C03653=1212.909,290.685,-66.684,-176.596,6.990,148.306
C03654=1212.913,290.437,-66.657,-176.598,6.987,148.306
C03655=1212.918,290.189,-66.627,-176.601,6.985,148.306
C03656=1212.922,289.941,-66.598,-176.603,6.983,148.306
C03657=1212.926,289.692,-66.569,-176.606,6.980,148.306
C03658=1212.931,289.418,-66.537,-176.609,6.977,148.306
C03659=1212.935,289.144,-66.505,-176.611,6.975,148.306
C03660=1212.940,288.869,-66.473,-176.614,6.972,148.306
C03661=1212.945,288.595,-66.442,-176.617,6.969,148.306
C03662=1212.950,288.347,-66.413,-176.619,6.967,148.306
C03663=1212.954,288.099,-66.384,-176.621,6.964,148.306
C03664=1212.958,287.851,-66.355,-176.624,6.962,148.307
C03665=1212.963,287.602,-66.327,-176.627,6.959,148.307
C03666=1212.967,287.354,-66.297,-176.629,6.957,148.307
C03667=1212.972,287.105,-66.268,-176.631,6.954,148.307
C03668=1212.976,286.858,-66.240,-176.634,6.952,148.307
C03669=1212.980,286.609,-66.211,-176.636,6.949,148.307
C03670=1212.985,286.360,-66.182,-176.639,6.946,148.307
C03671=1212.989,286.113,-66.154,-176.641,6.944,148.307
C03672=1212.993,285.864,-66.125,-176.644,6.941,148.307
C03673=1212.998,285.615,-66.096,-176.646,6.939,148.308
C03674=1213.002,285.368,-66.068,-176.648,6.937,148.308
C03675=1213.006,285.119,-66.039,-176.651,6.934,148.308
C03676=1213.011,284.870,-66.010,-176.654,6.932,148.308
C03677=1213.015,284.623,-65.982,-176.656,6.929,148.308
C03678=1213.019,284.374,-65.953,-176.658,6.927,148.308
C03679=1213.024,284.126,-65.925,-176.661,6.925,148.308
C03680=1213.028,283.878,-65.896,-176.664,6.922,148.308
C03681=1213.032,283.629,-65.867,-176.666,6.920,148.308
C03682=1213.037,283.381,-65.839,-176.668,6.918,148.308
C03683=1213.041,283.132,-65.811,-176.671,6.915,148.309
C03684=1213.045,282.884,-65.781,-176.673,6.913,148.309
C03685=1213.050,282.636,-65.754,-176.676,6.910,148.309
C03686=1213.054,282.387,-65.725,-176.679,6.908,148.309
C03687=1213.058,282.139,-65.697,-176.681,6.906,148.309
C03688=1213.063,281.890,-65.668,-176.683,6.903,148.309
C03689=1213.068,281.643,-65.639,-176.686,6.901,148.309
C03690=1213.071,281.394,-65.611,-176.689,6.898,148.309
C03691=1213.076,281.145,-65.582,-176.691,6.895,148.310
C03692=1213.080,280.898,-65.555,-176.693,6.894,148.310
C03693=1213.085,280.649,-65.526,-176.696,6.891,148.310
C03694=1213.089,280.401,-65.498,-176.698,6.888,148.310
C03695=1213.094,280.152,-65.469,-176.701,6.887,148.310
C03696=1213.098,279.905,-65.441,-176.704,6.883,148.310
C03697=1213.102,279.656,-65.412,-176.706,6.881,148.310
C03698=1213.106,279.408,-65.384,-176.709,6.879,148.311
C03699=1213.110,279.159,-65.356,-176.711,6.876,148.311
C03700=1213.115,278.911,-65.328,-176.713,6.874,148.311
C03701=1213.119,278.663,-65.300,-176.716,6.871,148.311
C03702=1213.124,278.414,-65.271,-176.718,6.869,148.311
C03703=1213.128,278.166,-65.243,-176.720,6.867,148.311
C03704=1213.132,277.917,-65.214,-176.724,6.864,148.311
C03705=1213.137,277.669,-65.187,-176.726,6.862,148.311
C03706=1213.141,277.420,-65.158,-176.728,6.860,148.311
C03707=1213.146,277.172,-65.130,-176.731,6.857,148.312
C03708=1213.149,276.924,-65.102,-176.733,6.855,148.312
C03709=1213.154,276.675,-65.074,-176.735,6.853,148.312
C03710=1213.159,276.428,-65.046,-176.738,6.850,148.312
C03711=1213.163,276.178,-65.018,-176.741,6.848,148.312
C03712=1213.168,275.930,-64.990,-176.744,6.845,148.312
C03713=1213.172,275.682,-64.962,-176.746,6.843,148.313
C03714=1213.177,275.433,-64.933,-176.748,6.841,148.313
C03715=1213.180,275.185,-64.905,-176.751,6.838,148.313
C03716=1213.185,274.937,-64.878,-176.753,6.836,148.313
C03717=1213.189,274.688,-64.849,-176.756,6.834,148.313
C03718=1213.194,274.440,-64.821,-176.759,6.831,148.313
C03719=1213.198,274.191,-64.794,-176.761,6.829,148.313
C03720=1213.202,273.943,-64.766,-176.763,6.827,148.314
C03721=1213.207,273.695,-64.737,-176.766,6.824,148.314
C03722=1213.211,273.446,-64.709,-176.769,6.822,148.314
C03723=1213.215,273.199,-64.682,-176.771,6.820,148.314
C03724=1213.220,272.949,-64.654,-176.773,6.817,148.314
C03725=1213.224,272.701,-64.626,-176.776,6.815,148.314
C03726=1213.228,272.453,-64.598,-176.778,6.813,148.314
C03727=1213.233,272.205,-64.570,-176.781,6.810,148.315
C03728=1213.238,271.956,-64.542,-176.784,6.808,148.315
C03729=1213.242,271.707,-64.514,-176.786,6.806,148.315
C03730=1213.246,271.459,-64.486,-176.788,6.804,148.315
C03731=1213.251,271.211,-64.459,-176.791,6.801,148.315
C03732=1213.255,270.962,-64.430,-176.794,6.799,148.315
C03733=1213.260,270.714,-64.403,-176.796,6.797,148.316
C03734=1213.264,270.465,-64.375,-176.799,6.794,148.316
C03735=1213.268,270.217,-64.347,-176.801,6.792,148.316
C03736=1213.272,269.969,-64.320,-176.804,6.790,148.316
C03737=1213.277,269.720,-64.292,-176.806,6.787,148.316
C03738=1213.281,269.472,-64.264,-176.808,6.785,148.316
C03739=1213.286,269.223,-64.237,-176.811,6.783,148.317
C03740=1213.290,268.975,-64.209,-176.814,6.780,148.317
C03741=1213.294,268.726,-64.182,-176.816,6.778,148.317
C03742=1213.299,268.478,-64.154,-176.818,6.776,148.317
C03743=1213.303,268.230,-64.126,-176.821,6.774,148.317
C03744=1213.308,267.981,-64.098,-176.824,6.771,148.317
C03745=1213.312,267.733,-64.070,-176.826,6.769,148.318
C03746=1213.316,267.484,-64.043,-176.829,6.767,148.318
C03747=1213.321,267.236,-64.015,-176.832,6.764,148.318
C03748=1213.325,266.988,-63.988,-176.834,6.762,148.318
C03749=1213.330,266.740,-63.960,-176.836,6.760,148.318
C03750=1213.334,266.491,-63.933,-176.839,6.758,148.318
C03751=1213.338,266.242,-63.906,-176.841,6.755,148.318
C03752=1213.343,265.994,-63.878,-176.844,6.753,148.319
C03753=1213.347,265.745,-63.851,-176.846,6.751,148.319
C03754=1213.351,265.497,-63.823,-176.849,6.748,148.319
C03755=1213.357,265.248,-63.795,-176.851,6.746,148.319
C03756=1213.361,265.000,-63.768,-176.854,6.744,148.319
C03757=1213.365,264.751,-63.740,-176.856,6.742,148.320
C03758=1213.370,264.503,-63.713,-176.859,6.739,148.320
C03759=1213.374,264.255,-63.685,-176.861,6.737,148.320
C03760=1213.379,264.006,-63.658,-176.864,6.735,148.320
C03761=1213.383,263.757,-63.631,-176.866,6.733,148.320
C03762=1213.387,263.485,-63.601,-176.869,6.730,148.321
C03763=1213.393,263.212,-63.571,-176.872,6.727,148.321
C03764=1213.397,262.940,-63.541,-176.875,6.725,148.321
C03765=1213.402,262.667,-63.511,-176.878,6.723,148.321
C03766=1213.406,262.418,-63.483,-176.880,6.721,148.321
C03767=1213.411,262.170,-63.456,-176.882,6.718,148.322
C03768=1213.416,261.921,-63.429,-176.886,6.716,148.322
C03769=1213.419,261.674,-63.402,-176.888,6.714,148.322
C03770=1213.424,261.425,-63.375,-176.890,6.712,148.322
C03771=1213.428,261.176,-63.347,-176.893,6.710,148.322
C03772=1213.433,260.927,-63.320,-176.896,6.707,148.323
C03773=1213.437,260.679,-63.292,-176.898,6.705,148.323
C03774=1213.442,260.431,-63.265,-176.900,6.703,148.323
C03775=1213.446,260.182,-63.238,-176.903,6.701,148.323
C03776=1213.450,259.933,-63.211,-176.906,6.698,148.323
C03777=1213.455,259.685,-63.184,-176.908,6.696,148.323
C03778=1213.459,259.437,-63.157,-176.910,6.694,148.324
C03779=1213.464,259.188,-63.130,-176.913,6.692,148.324
C03780=1213.468,258.940,-63.103,-176.915,6.690,148.324
C03781=1213.473,258.692,-63.075,-176.918,6.687,148.324
C03782=1213.477,258.443,-63.048,-176.921,6.685,148.324
C03783=1213.481,258.194,-63.021,-176.923,6.683,148.325
C03784=1213.485,257.946,-62.995,-176.925,6.681,148.325
C03785=1213.490,257.697,-62.967,-176.928,6.678,148.325
C03786=1213.495,257.449,-62.940,-176.931,6.676,148.325
C03787=1213.499,257.200,-62.913,-176.933,6.674,148.325
C03788=1213.504,256.952,-62.886,-176.936,6.672,148.326
C03789=1213.508,256.704,-62.860,-176.938,6.670,148.326
C03790=1213.512,256.455,-62.833,-176.941,6.667,148.326
C03791=1213.516,256.206,-62.805,-176.943,6.665,148.326
C03792=1213.521,255.957,-62.778,-176.946,6.663,148.326
C03793=1213.526,255.709,-62.751,-176.948,6.661,148.327
C03794=1213.530,255.461,-62.725,-176.951,6.658,148.327
C03795=1213.534,255.212,-62.698,-176.954,6.656,148.327
C03796=1213.539,254.964,-62.671,-176.956,6.654,148.327
C03797=1213.543,254.715,-62.645,-176.959,6.652,148.328
C03798=1213.548,254.467,-62.618,-176.961,6.650,148.328
C03799=1213.553,254.218,-62.591,-176.964,6.648,148.328
C03800=1213.557,253.970,-62.564,-176.967,6.646,148.328
C03801=1213.561,253.721,-62.537,-176.969,6.643,148.328
C03802=1213.566,253.473,-62.510,-176.971,6.642,148.329
C03803=1213.570,253.224,-62.483,-176.973,6.639,148.329
C03804=1213.574,252.976,-62.457,-176.977,6.637,148.329
C03805=1213.579,252.727,-62.430,-176.979,6.635,148.329
C03806=1213.584,252.479,-62.403,-176.981,6.633,148.329
C03807=1213.587,252.230,-62.376,-176.984,6.631,148.330
C03808=1213.592,251.981,-62.349,-176.986,6.629,148.330
C03809=1213.596,251.733,-62.323,-176.989,6.626,148.330
C03810=1213.601,251.484,-62.296,-176.992,6.624,148.330
C03811=1213.606,251.235,-62.269,-176.994,6.622,148.330
C03812=1213.609,250.987,-62.243,-176.997,6.620,148.331
C03813=1213.614,250.738,-62.217,-176.999,6.618,148.331
C03814=1213.618,250.490,-62.190,-177.001,6.616,148.331
C03815=1213.623,250.241,-62.163,-177.005,6.613,148.331
C03816=1213.628,249.993,-62.136,-177.007,6.611,148.331
C03817=1213.632,249.744,-62.110,-177.009,6.609,148.332
C03818=1213.637,249.496,-62.083,-177.012,6.607,148.332
C03819=1213.641,249.248,-62.057,-177.014,6.605,148.332
C03820=1213.646,248.999,-62.031,-177.017,6.603,148.332
C03821=1213.650,248.751,-62.004,-177.020,6.601,148.333
C03822=1213.655,248.502,-61.978,-177.022,6.598,148.333
C03823=1213.659,248.254,-61.951,-177.025,6.597,148.333
C03824=1213.663,248.005,-61.924,-177.027,6.595,148.333
C03825=1213.668,247.756,-61.899,-177.029,6.593,148.334
C03826=1213.672,247.508,-61.872,-177.032,6.591,148.334
C03827=1213.677,247.259,-61.846,-177.035,6.588,148.334
C03828=1213.681,247.010,-61.819,-177.037,6.586,148.334
C03829=1213.685,246.762,-61.792,-177.040,6.584,148.335
C03830=1213.690,246.513,-61.766,-177.042,6.582,148.335
C03831=1213.694,246.265,-61.740,-177.045,6.580,148.335
C03832=1213.699,246.016,-61.713,-177.047,6.578,148.335
C03833=1213.703,245.768,-61.687,-177.050,6.576,148.335
C03834=1213.708,245.519,-61.660,-177.053,6.573,148.336
C03835=1213.712,245.271,-61.634,-177.055,6.571,148.336
C03836=1213.717,245.022,-61.608,-177.057,6.569,148.336
C03837=1213.722,244.773,-61.582,-177.060,6.567,148.336
C03838=1213.725,244.525,-61.556,-177.063,6.565,148.337
C03839=1213.730,244.276,-61.529,-177.065,6.563,148.337
C03840=1213.734,244.028,-61.503,-177.067,6.561,148.337
C03841=1213.739,243.779,-61.477,-177.071,6.559,148.337
C03842=1213.743,243.530,-61.450,-177.073,6.557,148.338
C03843=1213.748,243.282,-61.425,-177.075,6.555,148.338
C03844=1213.753,243.033,-61.398,-177.078,6.553,148.338
C03845=1213.757,242.785,-61.372,-177.081,6.551,148.338
C03846=1213.761,242.536,-61.346,-177.083,6.549,148.338
C03847=1213.766,242.287,-61.320,-177.085,6.547,148.339
C03848=1213.770,242.039,-61.293,-177.088,6.545,148.339
C03849=1213.774,241.790,-61.268,-177.091,6.542,148.339
C03850=1213.780,241.542,-61.242,-177.093,6.540,148.339
C03851=1213.784,241.293,-61.215,-177.096,6.538,148.340
C03852=1213.788,241.045,-61.189,-177.098,6.536,148.340
C03853=1213.793,240.795,-61.163,-177.101,6.534,148.340
C03854=1213.797,240.547,-61.137,-177.103,6.532,148.341
C03855=1213.802,240.299,-61.111,-177.106,6.530,148.341
C03856=1213.806,240.050,-61.085,-177.108,6.528,148.341
C03857=1213.811,239.801,-61.059,-177.111,6.526,148.341
C03858=1213.815,239.552,-61.033,-177.114,6.524,148.342
C03859=1213.819,239.304,-61.007,-177.116,6.522,148.342
C03860=1213.824,239.056,-60.981,-177.119,6.520,148.342
C03861=1213.829,238.807,-60.955,-177.121,6.518,148.342
C03862=1213.833,238.558,-60.929,-177.124,6.516,148.343
C03863=1213.837,238.309,-60.904,-177.126,6.514,148.343
C03864=1213.842,238.061,-60.878,-177.129,6.512,148.343
C03865=1213.847,237.813,-60.851,-177.131,6.510,148.343
C03866=1213.851,237.541,-60.823,-177.135,6.507,148.344
C03867=1213.857,237.270,-60.795,-177.137,6.506,148.344
C03868=1213.861,236.999,-60.767,-177.140,6.503,148.344
C03869=1213.866,236.727,-60.739,-177.143,6.501,148.344
C03870=1213.871,236.478,-60.713,-177.145,6.499,148.345
C03871=1213.875,236.230,-60.688,-177.148,6.497,148.345
C03872=1213.879,235.981,-60.662,-177.150,6.495,148.345
C03873=1213.884,235.732,-60.635,-177.153,6.493,148.345
C03874=1213.889,235.484,-60.610,-177.155,6.491,148.346
C03875=1213.893,235.235,-60.584,-177.158,6.489,148.346
C03876=1213.897,234.986,-60.559,-177.160,6.487,148.346
C03877=1213.902,234.738,-60.533,-177.163,6.484,148.346
C03878=1213.906,234.489,-60.507,-177.166,6.482,148.347
C03879=1213.911,234.240,-60.482,-177.168,6.481,148.347
C03880=1213.915,233.992,-60.456,-177.171,6.479,148.347
C03881=1213.920,233.743,-60.431,-177.173,6.477,148.347
C03882=1213.925,233.494,-60.404,-177.176,6.475,148.348
C03883=1213.929,233.246,-60.378,-177.178,6.473,148.348
C03884=1213.934,232.997,-60.353,-177.181,6.471,148.348
C03885=1213.938,232.749,-60.327,-177.184,6.469,148.349
C03886=1213.942,232.500,-60.302,-177.186,6.467,148.349
C03887=1213.947,232.252,-60.276,-177.188,6.465,148.349
C03888=1213.951,232.003,-60.250,-177.191,6.463,148.349
C03889=1213.956,231.753,-60.225,-177.194,6.461,148.350
C03890=1213.961,231.505,-60.200,-177.196,6.459,148.350
C03891=1213.965,231.257,-60.174,-177.199,6.457,148.350
C03892=1213.970,231.008,-60.149,-177.202,6.455,148.350
C03893=1213.974,230.760,-60.123,-177.204,6.453,148.351
C03894=1213.978,230.511,-60.097,-177.207,6.451,148.351
C03895=1213.983,230.262,-60.073,-177.209,6.449,148.351
C03896=1213.987,230.013,-60.047,-177.212,6.447,148.352
C03897=1213.992,229.765,-60.021,-177.214,6.445,148.352
C03898=1213.996,229.516,-59.996,-177.217,6.443,148.352
C03899=1214.001,229.267,-59.971,-177.220,6.441,148.352
C03900=1214.006,229.019,-59.945,-177.222,6.439,148.353
C03901=1214.010,228.770,-59.920,-177.224,6.437,148.353
C03902=1214.014,228.521,-59.894,-177.227,6.436,148.353
C03903=1214.019,228.273,-59.869,-177.230,6.434,148.354
C03904=1214.023,228.024,-59.844,-177.232,6.432,148.354
C03905=1214.028,227.776,-59.819,-177.235,6.430,148.354
C03906=1214.032,227.527,-59.794,-177.237,6.428,148.354
C03907=1214.037,227.278,-59.768,-177.240,6.426,148.355
C03908=1214.041,227.030,-59.743,-177.242,6.424,148.355
C03909=1214.046,226.780,-59.717,-177.245,6.422,148.355
C03910=1214.051,226.532,-59.692,-177.248,6.420,148.356
C03911=1214.055,226.283,-59.666,-177.250,6.418,148.356
C03912=1214.059,226.035,-59.642,-177.253,6.416,148.356
C03913=1214.063,225.786,-59.617,-177.256,6.414,148.356
C03914=1214.069,225.537,-59.592,-177.258,6.412,148.357
C03915=1214.073,225.289,-59.566,-177.261,6.410,148.357
C03916=1214.078,225.040,-59.541,-177.263,6.408,148.357
C03917=1214.082,224.791,-59.516,-177.266,6.406,148.357
C03918=1214.086,224.543,-59.491,-177.268,6.404,148.358
C03919=1214.091,224.294,-59.466,-177.271,6.402,148.358
C03920=1214.096,224.046,-59.440,-177.273,6.400,148.358
C03921=1214.100,223.796,-59.415,-177.276,6.399,148.359
C03922=1214.105,223.548,-59.390,-177.279,6.397,148.359
C03923=1214.109,223.299,-59.366,-177.281,6.395,148.359
C03924=1214.114,223.051,-59.340,-177.284,6.393,148.359
C03925=1214.118,222.802,-59.315,-177.286,6.391,148.360
C03926=1214.123,222.553,-59.290,-177.289,6.389,148.360
C03927=1214.127,222.304,-59.265,-177.291,6.387,148.360
C03928=1214.132,222.056,-59.241,-177.294,6.385,148.361
C03929=1214.136,221.807,-59.215,-177.297,6.383,148.361
C03930=1214.141,221.558,-59.190,-177.299,6.382,148.361
C03931=1214.145,221.310,-59.165,-177.301,6.379,148.362
C03932=1214.150,221.061,-59.140,-177.304,6.378,148.362
C03933=1214.154,220.811,-59.115,-177.307,6.376,148.362
C03934=1214.158,220.564,-59.091,-177.309,6.374,148.363
C03935=1214.163,220.314,-59.066,-177.312,6.372,148.363
C03936=1214.168,220.066,-59.040,-177.315,6.370,148.363
C03937=1214.172,219.818,-59.016,-177.317,6.368,148.364
C03938=1214.177,219.568,-58.991,-177.320,6.366,148.364
C03939=1214.182,219.320,-58.966,-177.322,6.364,148.364
C03940=1214.185,219.071,-58.941,-177.325,6.362,148.364
C03941=1214.191,218.822,-58.917,-177.327,6.361,148.365
C03942=1214.195,218.573,-58.892,-177.330,6.359,148.365
C03943=1214.199,218.325,-58.867,-177.333,6.357,148.365
C03944=1214.204,218.076,-58.842,-177.335,6.355,148.366
C03945=1214.209,217.827,-58.817,-177.338,6.353,148.366
C03946=1214.213,217.579,-58.793,-177.341,6.351,148.366
C03947=1214.217,217.330,-58.767,-177.343,6.350,148.367
C03948=1214.222,217.081,-58.743,-177.346,6.348,148.367
C03949=1214.227,216.833,-58.718,-177.348,6.346,148.367
C03950=1214.231,216.583,-58.693,-177.351,6.344,148.367
C03951=1214.236,216.335,-58.669,-177.353,6.342,148.368
C03952=1214.241,216.087,-58.644,-177.356,6.340,148.368
C03953=1214.244,215.838,-58.620,-177.358,6.338,148.368
C03954=1214.250,215.589,-58.595,-177.361,6.336,148.369
C03955=1214.254,215.340,-58.571,-177.364,6.334,148.369
C03956=1214.259,215.091,-58.546,-177.366,6.333,148.369
C03957=1214.263,214.843,-58.522,-177.369,6.331,148.370
C03958=1214.267,214.593,-58.497,-177.372,6.329,148.370
C03959=1214.272,214.345,-58.473,-177.374,6.327,148.370
C03960=1214.277,214.096,-58.448,-177.377,6.325,148.371
C03961=1214.280,213.848,-58.423,-177.380,6.323,148.371
C03962=1214.286,213.599,-58.398,-177.382,6.321,148.371
C03963=1214.290,213.350,-58.374,-177.384,6.319,148.371
C03964=1214.295,213.102,-58.349,-177.387,6.318,148.372
C03965=1214.299,212.853,-58.325,-177.390,6.316,148.372
C03966=1214.304,212.604,-58.300,-177.392,6.314,148.372
C03967=1214.308,212.355,-58.276,-177.395,6.312,148.373
C03968=1214.313,212.106,-58.251,-177.398,6.310,148.373
C03969=1214.317,211.858,-58.227,-177.400,6.308,148.373
C03970=1214.323,211.587,-58.201,-177.403,6.306,148.374
C03971=1214.328,211.317,-58.174,-177.405,6.305,148.374
C03972=1214.333,211.046,-58.147,-177.408,6.303,148.375
C03973=1214.337,210.776,-58.121,-177.412,6.300,148.375
C03974=1214.342,210.527,-58.096,-177.414,6.298,148.375
C03975=1214.346,210.279,-58.072,-177.416,6.297,148.376
C03976=1214.351,210.029,-58.049,-177.419,6.295,148.376
C03977=1214.356,209.780,-58.024,-177.421,6.294,148.376
C03978=1214.360,209.532,-58.000,-177.424,6.292,148.377
C03979=1214.365,209.283,-57.975,-177.427,6.290,148.377
C03980=1214.369,209.034,-57.951,-177.429,6.288,148.377
C03981=1214.373,208.786,-57.927,-177.432,6.286,148.378
C03982=1214.379,208.537,-57.902,-177.435,6.284,148.378
C03983=1214.383,208.288,-57.879,-177.437,6.283,148.378
C03984=1214.388,208.039,-57.855,-177.440,6.281,148.379
C03985=1214.392,207.790,-57.830,-177.442,6.279,148.379
C03986=1214.397,207.542,-57.806,-177.445,6.277,148.379
C03987=1214.401,207.293,-57.781,-177.448,6.275,148.380
C03988=1214.406,207.044,-57.758,-177.450,6.273,148.380
C03989=1214.411,206.795,-57.733,-177.453,6.271,148.380
C03990=1214.415,206.546,-57.709,-177.456,6.270,148.381
C03991=1214.419,206.298,-57.685,-177.458,6.268,148.381
C03992=1214.424,206.049,-57.661,-177.460,6.267,148.381
C03993=1214.429,205.800,-57.637,-177.463,6.265,148.382
C03994=1214.433,205.552,-57.613,-177.466,6.263,148.382
C03995=1214.438,205.303,-57.589,-177.468,6.261,148.382
C03996=1214.442,205.053,-57.564,-177.471,6.259,148.383
C03997=1214.447,204.805,-57.540,-177.474,6.258,148.383
C03998=1214.452,204.556,-57.517,-177.476,6.256,148.383
C03999=1214.456,204.307,-57.493,-177.479,6.254,148.384
C04000=1214.461,204.059,-57.468,-177.482,6.252,148.384
C04001=1214.466,203.810,-57.445,-177.484,6.250,148.384
C04002=1214.470,203.561,-57.420,-177.487,6.248,148.385
C04003=1214.474,203.312,-57.396,-177.489,6.247,148.385
C04004=1214.479,203.063,-57.373,-177.492,6.246,148.385
C04005=1214.483,202.815,-57.349,-177.494,6.244,148.386
C04006=1214.488,202.565,-57.325,-177.497,6.242,148.386
C04007=1214.493,202.317,-57.301,-177.499,6.240,148.386
C04008=1214.498,202.068,-57.278,-177.502,6.238,148.387
C04009=1214.502,201.820,-57.253,-177.505,6.236,148.387
C04010=1214.506,201.570,-57.230,-177.507,6.235,148.387
C04011=1214.510,201.321,-57.206,-177.510,6.233,148.388
C04012=1214.515,201.073,-57.182,-177.513,6.231,148.388
C04013=1214.520,200.824,-57.158,-177.515,6.230,148.388
C04014=1214.525,200.575,-57.134,-177.517,6.228,148.389
C04015=1214.529,200.326,-57.110,-177.520,6.226,148.389
C04016=1214.534,200.077,-57.087,-177.523,6.224,148.390
C04017=1214.538,199.829,-57.063,-177.525,6.223,148.390
C04018=1214.543,199.580,-57.039,-177.528,6.221,148.390
C04019=1214.548,199.331,-57.015,-177.531,6.219,148.391
C04020=1214.552,199.082,-56.992,-177.533,6.217,148.391
C04021=1214.557,198.834,-56.968,-177.536,6.215,148.391
C04022=1214.561,198.585,-56.945,-177.538,6.214,148.392
C04023=1214.566,198.336,-56.921,-177.541,6.212,148.392
C04024=1214.570,198.087,-56.897,-177.543,6.211,148.392
C04025=1214.575,197.838,-56.873,-177.546,6.209,148.393
C04026=1214.579,197.589,-56.850,-177.549,6.207,148.393
C04027=1214.584,197.340,-56.826,-177.551,6.205,148.393
C04028=1214.588,197.091,-56.803,-177.554,6.203,148.394
C04029=1214.593,196.843,-56.779,-177.557,6.201,148.394
C04030=1214.597,196.594,-56.755,-177.559,6.200,148.394
C04031=1214.602,196.345,-56.732,-177.561,6.199,148.395
C04032=1214.607,196.096,-56.708,-177.564,6.197,148.395
C04033=1214.611,195.847,-56.684,-177.567,6.195,148.395
C04034=1214.616,195.598,-56.661,-177.570,6.193,148.396
C04035=1214.621,195.349,-56.638,-177.572,6.192,148.396
C04036=1214.625,195.100,-56.614,-177.575,6.190,148.397
C04037=1214.630,194.852,-56.590,-177.577,6.189,148.397
C04038=1214.634,194.603,-56.567,-177.580,6.187,148.397
C04039=1214.639,194.354,-56.544,-177.582,6.185,148.398
C04040=1214.644,194.105,-56.521,-177.585,6.183,148.398
C04041=1214.649,193.857,-56.496,-177.588,6.181,148.398
C04042=1214.654,193.608,-56.473,-177.590,6.180,148.399
C04043=1214.658,193.359,-56.450,-177.592,6.179,148.399
C04044=1214.663,193.110,-56.426,-177.595,6.177,148.400
C04045=1214.667,192.861,-56.404,-177.598,6.175,148.400
C04046=1214.672,192.612,-56.380,-177.600,6.173,148.400
C04047=1214.676,192.364,-56.356,-177.603,6.171,148.401
C04048=1214.681,192.115,-56.333,-177.606,6.169,148.401
C04049=1214.685,191.866,-56.309,-177.608,6.168,148.401
C04050=1214.690,191.617,-56.286,-177.611,6.167,148.402
C04051=1214.695,191.368,-56.263,-177.614,6.165,148.402
C04052=1214.699,191.118,-56.239,-177.616,6.163,148.403
C04053=1214.703,190.870,-56.217,-177.619,6.161,148.403
C04054=1214.708,190.621,-56.193,-177.621,6.160,148.403
C04055=1214.713,190.372,-56.170,-177.624,6.159,148.404
C04056=1214.718,190.123,-56.147,-177.626,6.157,148.404
C04057=1214.723,189.874,-56.124,-177.629,6.155,148.404
C04058=1214.727,189.626,-56.101,-177.631,6.153,148.405
C04059=1214.732,189.377,-56.077,-177.634,6.151,148.405
C04060=1214.736,189.128,-56.054,-177.637,6.149,148.405
C04061=1214.741,188.879,-56.031,-177.639,6.148,148.406
C04062=1214.746,188.629,-56.007,-177.642,6.147,148.406
C04063=1214.750,188.381,-55.985,-177.645,6.145,148.407
C04064=1214.755,188.132,-55.962,-177.647,6.143,148.407
C04065=1214.760,187.883,-55.938,-177.650,6.141,148.407
C04066=1214.764,187.635,-55.915,-177.652,6.140,148.408
C04067=1214.768,187.386,-55.892,-177.655,6.139,148.408
C04068=1214.773,187.137,-55.869,-177.657,6.137,148.408
C04069=1214.778,186.888,-55.845,-177.660,6.135,148.409
C04070=1214.782,186.640,-55.823,-177.663,6.133,148.409
C04071=1214.787,186.391,-55.800,-177.665,6.132,148.410
C04072=1214.792,186.141,-55.777,-177.668,6.131,148.410
C04073=1214.796,185.892,-55.754,-177.671,6.129,148.410
C04074=1214.801,185.622,-55.729,-177.673,6.127,148.411
C04075=1214.807,185.353,-55.704,-177.676,6.125,148.411
C04076=1214.811,185.083,-55.680,-177.679,6.124,148.412
C04077=1214.816,184.814,-55.654,-177.682,6.122,148.412
C04078=1214.821,184.564,-55.631,-177.684,6.120,148.412
C04079=1214.825,184.316,-55.609,-177.687,6.118,148.413
C04080=1214.830,184.067,-55.586,-177.689,6.117,148.413
C04081=1214.835,183.818,-55.562,-177.692,6.115,148.414
C04082=1214.839,183.569,-55.540,-177.694,6.114,148.414
C04083=1214.844,183.320,-55.517,-177.697,6.112,148.414
C04084=1214.849,183.072,-55.494,-177.700,6.111,148.415
C04085=1214.853,182.823,-55.471,-177.702,6.109,148.415
C04086=1214.858,182.573,-55.448,-177.705,6.107,148.416
C04087=1214.862,182.324,-55.426,-177.708,6.106,148.416
C04088=1214.867,182.075,-55.402,-177.710,6.104,148.416
C04089=1214.872,181.827,-55.380,-177.712,6.103,148.417
C04090=1214.877,181.578,-55.357,-177.715,6.101,148.417
C04091=1214.880,181.329,-55.334,-177.718,6.099,148.418
C04092=1214.886,181.081,-55.311,-177.721,6.098,148.418
C04093=1214.890,180.831,-55.289,-177.723,6.097,148.418
C04094=1214.895,180.582,-55.266,-177.725,6.095,148.419
C04095=1214.899,180.333,-55.244,-177.728,6.093,148.419
C04096=1214.904,180.085,-55.221,-177.731,6.091,148.419
C04097=1214.909,179.836,-55.198,-177.733,6.090,148.420
C04098=1214.913,179.586,-55.176,-177.736,6.089,148.420
C04099=1214.918,179.337,-55.152,-177.739,6.087,148.421
C04100=1214.923,179.089,-55.131,-177.741,6.085,148.421
C04101=1214.927,178.840,-55.108,-177.743,6.084,148.421
C04102=1214.932,178.590,-55.085,-177.746,6.082,148.422
C04103=1214.936,178.342,-55.063,-177.749,6.080,148.422
C04104=1214.941,178.093,-55.039,-177.752,6.079,148.423
C04105=1214.945,177.844,-55.017,-177.754,6.078,148.423
C04106=1214.951,177.596,-54.994,-177.757,6.076,148.423
C04107=1214.955,177.346,-54.972,-177.759,6.074,148.424
C04108=1214.960,177.097,-54.949,-177.762,6.072,148.424
C04109=1214.965,176.849,-54.927,-177.764,6.071,148.425
C04110=1214.969,176.599,-54.904,-177.767,6.070,148.425
C04111=1214.973,176.350,-54.882,-177.770,6.068,148.426
C04112=1214.978,176.102,-54.860,-177.772,6.067,148.426
C04113=1214.983,175.852,-54.837,-177.775,6.065,148.426
C04114=1214.987,175.603,-54.815,-177.777,6.064,148.427
C04115=1214.993,175.355,-54.792,-177.780,6.062,148.427
C04116=1214.997,175.105,-54.770,-177.783,6.061,148.428
C04117=1215.001,174.857,-54.747,-177.785,6.059,148.428
C04118=1215.006,174.608,-54.725,-177.788,6.057,148.428
C04119=1215.011,174.358,-54.703,-177.790,6.056,148.429
C04120=1215.015,174.110,-54.680,-177.793,6.055,148.429
C04121=1215.020,173.861,-54.658,-177.796,6.053,148.430
C04122=1215.025,173.611,-54.636,-177.798,6.051,148.430
C04123=1215.029,173.363,-54.613,-177.800,6.050,148.430
C04124=1215.034,173.114,-54.591,-177.803,6.048,148.431
C04125=1215.039,172.865,-54.569,-177.806,6.047,148.431
C04126=1215.043,172.616,-54.546,-177.808,6.046,148.432
C04127=1215.049,172.367,-54.524,-177.811,6.044,148.432
C04128=1215.053,172.118,-54.502,-177.814,6.042,148.432
C04129=1215.057,171.869,-54.480,-177.816,6.041,148.433
C04130=1215.062,171.620,-54.457,-177.818,6.040,148.433
C04131=1215.067,171.371,-54.435,-177.822,6.038,148.434
C04132=1215.072,171.122,-54.413,-177.824,6.036,148.434
C04133=1215.076,170.873,-54.391,-177.826,6.035,148.435
C04134=1215.081,170.625,-54.368,-177.829,6.033,148.435
C04135=1215.085,170.375,-54.346,-177.832,6.032,148.435
C04136=1215.090,170.127,-54.324,-177.834,6.031,148.436
C04137=1215.095,169.877,-54.302,-177.837,6.029,148.436
C04138=1215.100,169.628,-54.280,-177.840,6.027,148.437
C04139=1215.104,169.380,-54.257,-177.842,6.026,148.437
C04140=1215.108,169.130,-54.235,-177.844,6.025,148.437
C04141=1215.113,168.882,-54.213,-177.847,6.023,148.438
C04142=1215.118,168.632,-54.191,-177.850,6.021,148.438
C04143=1215.123,168.384,-54.169,-177.852,6.020,148.439
C04144=1215.127,168.134,-54.147,-177.855,6.018,148.439
C04145=1215.132,167.886,-54.125,-177.858,6.017,148.440
C04146=1215.136,167.636,-54.103,-177.860,6.016,148.440
C04147=1215.141,167.388,-54.081,-177.863,6.014,148.440
C04148=1215.146,167.139,-54.058,-177.865,6.012,148.441
C04149=1215.151,166.890,-54.037,-177.868,6.011,148.441
C04150=1215.155,166.641,-54.015,-177.871,6.010,148.442
C04151=1215.160,166.392,-53.993,-177.873,6.008,148.442
C04152=1215.164,166.143,-53.971,-177.875,6.007,148.442
C04153=1215.169,165.894,-53.949,-177.878,6.005,148.443
C04154=1215.173,165.645,-53.927,-177.881,6.004,148.443
C04155=1215.178,165.396,-53.905,-177.883,6.003,148.444
C04156=1215.184,165.147,-53.883,-177.886,6.001,148.444
C04157=1215.188,164.898,-53.861,-177.889,5.999,148.445
C04158=1215.193,164.649,-53.839,-177.891,5.999,148.445
C04159=1215.197,164.400,-53.817,-177.894,5.997,148.446
C04160=1215.202,164.151,-53.796,-177.896,5.996,148.446
C04161=1215.206,163.902,-53.774,-177.899,5.994,148.446
C04162=1215.211,163.653,-53.752,-177.902,5.992,148.447
C04163=1215.216,163.404,-53.730,-177.904,5.991,148.447
C04164=1215.220,163.155,-53.708,-177.907,5.990,148.448
C04165=1215.226,162.906,-53.687,-177.909,5.988,148.448
C04166=1215.230,162.656,-53.665,-177.912,5.987,148.449
C04167=1215.235,162.408,-53.643,-177.915,5.985,148.449
C04168=1215.239,162.158,-53.621,-177.917,5.984,148.449
C04169=1215.244,161.910,-53.600,-177.919,5.983,148.450
C04170=1215.249,161.661,-53.578,-177.922,5.981,148.450
C04171=1215.253,161.412,-53.556,-177.925,5.979,148.451
C04172=1215.258,161.163,-53.535,-177.927,5.978,148.451
C04173=1215.263,160.913,-53.513,-177.930,5.977,148.452
C04174=1215.267,160.665,-53.491,-177.933,5.976,148.452
C04175=1215.272,160.416,-53.470,-177.935,5.974,148.452
C04176=1215.277,160.167,-53.448,-177.938,5.972,148.453
C04177=1215.282,159.917,-53.427,-177.940,5.972,148.453
C04178=1215.287,159.649,-53.403,-177.943,5.970,148.454
C04179=1215.292,159.380,-53.380,-177.946,5.968,148.454
C04180=1215.297,159.110,-53.356,-177.949,5.967,148.455
C04181=1215.302,158.842,-53.333,-177.952,5.965,148.455
C04182=1215.307,158.593,-53.312,-177.954,5.964,148.456
C04183=1215.311,158.343,-53.290,-177.957,5.962,148.456
C04184=1215.316,158.095,-53.268,-177.959,5.961,148.457
C04185=1215.321,157.846,-53.247,-177.962,5.960,148.457
C04186=1215.325,157.596,-53.225,-177.965,5.958,148.457
C04187=1215.330,157.347,-53.204,-177.967,5.957,148.458
C04188=1215.335,157.099,-53.182,-177.970,5.955,148.458
C04189=1215.340,156.849,-53.161,-177.972,5.955,148.459
C04190=1215.344,156.600,-53.139,-177.975,5.953,148.459
C04191=1215.349,156.352,-53.118,-177.977,5.951,148.460
C04192=1215.353,156.102,-53.096,-177.980,5.950,148.460
C04193=1215.358,155.853,-53.075,-177.983,5.949,148.461
C04194=1215.363,155.604,-53.054,-177.985,5.948,148.461
C04195=1215.368,155.355,-53.032,-177.988,5.946,148.462
C04196=1215.372,155.106,-53.010,-177.991,5.944,148.462
C04197=1215.377,154.857,-52.990,-177.993,5.943,148.462
C04198=1215.382,154.608,-52.968,-177.995,5.941,148.463
C04199=1215.386,154.358,-52.947,-177.998,5.941,148.463
C04200=1215.391,154.110,-52.925,-178.001,5.939,148.464
C04201=1215.396,153.860,-52.904,-178.003,5.937,148.464
C04202=1215.400,153.612,-52.883,-178.006,5.937,148.465
C04203=1215.405,153.362,-52.862,-178.009,5.935,148.465
C04204=1215.410,153.114,-52.840,-178.011,5.934,148.465
C04205=1215.415,152.864,-52.819,-178.014,5.932,148.466
C04206=1215.419,152.616,-52.798,-178.017,5.931,148.466
C04207=1215.424,152.366,-52.777,-178.019,5.930,148.467
C04208=1215.429,152.117,-52.755,-178.022,5.928,148.467
C04209=1215.434,151.868,-52.734,-178.024,5.927,148.468
C04210=1215.438,151.620,-52.713,-178.027,5.925,148.468
C04211=1215.443,151.370,-52.692,-178.029,5.925,148.469
C04212=1215.447,151.121,-52.670,-178.032,5.923,148.469
C04213=1215.453,150.872,-52.649,-178.034,5.922,148.470
C04214=1215.457,150.623,-52.628,-178.037,5.920,148.470
C04215=1215.462,150.374,-52.607,-178.040,5.919,148.471
C04216=1215.467,150.125,-52.586,-178.042,5.918,148.471
C04217=1215.471,149.876,-52.564,-178.045,5.916,148.472
C04218=1215.476,149.627,-52.543,-178.047,5.915,148.472
C04219=1215.481,149.377,-52.522,-178.050,5.913,148.472
C04220=1215.485,149.129,-52.501,-178.052,5.913,148.473
C04221=1215.490,148.880,-52.480,-178.055,5.911,148.473
C04222=1215.495,148.630,-52.459,-178.058,5.909,148.474
C04223=1215.499,148.382,-52.438,-178.060,5.909,148.474
C04224=1215.504,148.132,-52.417,-178.063,5.907,148.475
C04225=1215.509,147.883,-52.396,-178.065,5.906,148.475
C04226=1215.513,147.635,-52.375,-178.068,5.904,148.476
C04227=1215.519,147.386,-52.354,-178.070,5.903,148.476
C04228=1215.524,147.136,-52.333,-178.073,5.901,148.476
C04229=1215.528,146.887,-52.312,-178.076,5.901,148.477
C04230=1215.532,146.638,-52.291,-178.078,5.899,148.477
C04231=1215.537,146.389,-52.270,-178.080,5.898,148.478
C04232=1215.542,146.140,-52.249,-178.084,5.897,148.478
C04233=1215.547,145.891,-52.229,-178.086,5.896,148.479
C04234=1215.551,145.642,-52.207,-178.089,5.894,148.479
C04235=1215.557,145.393,-52.186,-178.092,5.892,148.480
C04236=1215.560,145.143,-52.165,-178.094,5.891,148.480
C04237=1215.566,144.894,-52.144,-178.097,5.890,148.481
C04238=1215.570,144.645,-52.124,-178.099,5.889,148.481
C04239=1215.575,144.396,-52.103,-178.102,5.887,148.482
C04240=1215.579,144.147,-52.082,-178.104,5.887,148.482
C04241=1215.584,143.898,-52.061,-178.107,5.885,148.483
C04242=1215.589,143.649,-52.041,-178.109,5.884,148.483
C04243=1215.594,143.400,-52.020,-178.112,5.882,148.484
C04244=1215.599,143.151,-51.999,-178.114,5.881,148.484
C04245=1215.604,142.902,-51.978,-178.117,5.880,148.485
C04246=1215.608,142.653,-51.958,-178.120,5.879,148.485
C04247=1215.613,142.404,-51.937,-178.122,5.877,148.485
C04248=1215.617,142.154,-51.916,-178.125,5.876,148.486
C04249=1215.622,141.905,-51.895,-178.127,5.875,148.486
C04250=1215.626,141.656,-51.874,-178.130,5.874,148.487
C04251=1215.632,141.407,-51.853,-178.133,5.872,148.487
C04252=1215.636,141.158,-51.833,-178.135,5.871,148.488
C04253=1215.641,140.909,-51.812,-178.138,5.870,148.488
C04254=1215.646,140.660,-51.792,-178.140,5.869,148.489
C04255=1215.650,140.411,-51.771,-178.143,5.867,148.489
C04256=1215.655,140.162,-51.750,-178.145,5.866,148.490
C04257=1215.660,139.913,-51.730,-178.148,5.865,148.490
C04258=1215.665,139.663,-51.709,-178.151,5.864,148.491
C04259=1215.669,139.415,-51.689,-178.153,5.862,148.491
C04260=1215.674,139.166,-51.668,-178.155,5.861,148.492
C04261=1215.679,138.916,-51.647,-178.159,5.860,148.492
C04262=1215.684,138.667,-51.628,-178.161,5.859,148.493
C04263=1215.689,138.417,-51.607,-178.164,5.857,148.493
C04264=1215.693,138.169,-51.586,-178.166,5.856,148.494
C04265=1215.698,137.920,-51.566,-178.169,5.855,148.494
C04266=1215.703,137.670,-51.545,-178.171,5.854,148.495
C04267=1215.707,137.421,-51.525,-178.174,5.852,148.495
C04268=1215.712,137.172,-51.504,-178.177,5.852,148.496
C04269=1215.717,136.923,-51.483,-178.179,5.850,148.496
C04270=1215.721,136.674,-51.463,-178.181,5.849,148.497
C04271=1215.726,136.425,-51.443,-178.185,5.847,148.497
C04272=1215.731,136.175,-51.422,-178.187,5.846,148.498
C04273=1215.736,135.926,-51.402,-178.190,5.845,148.498
C04274=1215.740,135.678,-51.381,-178.192,5.844,148.499
C04275=1215.745,135.428,-51.360,-178.195,5.843,148.499
C04276=1215.750,135.179,-51.340,-178.197,5.842,148.500
C04277=1215.755,134.930,-51.321,-178.199,5.841,148.500
C04278=1215.760,134.681,-51.300,-178.202,5.839,148.501
C04279=1215.765,134.432,-51.279,-178.205,5.838,148.501
C04280=1215.769,134.183,-51.259,-178.208,5.837,148.502
C04281=1215.774,133.934,-51.239,-178.210,5.836,148.502
C04282=1215.779,133.665,-51.217,-178.213,5.834,148.503
C04283=1215.784,133.396,-51.195,-178.216,5.832,148.503
C04284=1215.789,133.128,-51.173,-178.218,5.832,148.504
C04285=1215.795,132.859,-51.152,-178.222,5.830,148.504
C04286=1215.799,132.610,-51.131,-178.224,5.829,148.505
C04287=1215.803,132.361,-51.111,-178.226,5.828,148.505
C04288=1215.808,132.111,-51.091,-178.229,5.827,148.506
C04289=1215.814,131.863,-51.071,-178.232,5.825,148.506
C04290=1215.818,131.614,-51.050,-178.234,5.825,148.507
C04291=1215.823,131.364,-51.030,-178.237,5.823,148.507
C04292=1215.828,131.115,-51.010,-178.239,5.822,148.508
C04293=1215.832,130.866,-50.990,-178.242,5.820,148.508
C04294=1215.838,130.616,-50.969,-178.245,5.820,148.509
C04295=1215.842,130.367,-50.949,-178.247,5.819,148.509
C04296=1215.847,130.119,-50.929,-178.250,5.817,148.509
C04297=1215.852,129.870,-50.909,-178.252,5.816,148.510
C04298=1215.856,129.621,-50.889,-178.255,5.815,148.511
C04299=1215.861,129.371,-50.869,-178.257,5.814,148.511
C04300=1215.865,129.122,-50.849,-178.260,5.812,148.512
C04301=1215.871,128.872,-50.829,-178.263,5.812,148.512
C04302=1215.875,128.623,-50.808,-178.265,5.811,148.513
C04303=1215.881,128.374,-50.789,-178.268,5.809,148.513
C04304=1215.885,128.126,-50.769,-178.270,5.808,148.514
C04305=1215.890,127.877,-50.748,-178.273,5.807,148.514
C04306=1215.894,127.627,-50.729,-178.275,5.806,148.515
C04307=1215.899,127.378,-50.708,-178.279,5.804,148.515
C04308=1215.904,127.129,-50.689,-178.281,5.803,148.516
C04309=1215.908,126.880,-50.669,-178.283,5.802,148.516
C04310=1215.913,126.631,-50.649,-178.286,5.801,148.517
C04311=1215.918,126.381,-50.629,-178.288,5.800,148.517
C04312=1215.922,126.132,-50.609,-178.291,5.799,148.518
C04313=1215.928,125.883,-50.590,-178.293,5.798,148.518
C04314=1215.933,125.634,-50.569,-178.296,5.797,148.519
C04315=1215.938,125.384,-50.549,-178.299,5.795,148.519
C04316=1215.942,125.136,-50.529,-178.301,5.795,148.520
C04317=1215.947,124.886,-50.509,-178.304,5.793,148.520
C04318=1215.952,124.637,-50.490,-178.307,5.792,148.521
C04319=1215.957,124.388,-50.469,-178.309,5.791,148.521
C04320=1215.961,124.139,-50.450,-178.312,5.790,148.522
C04321=1215.966,123.890,-50.429,-178.314,5.789,148.522
C04322=1215.971,123.641,-50.410,-178.317,5.787,148.523
C04323=1215.976,123.391,-50.390,-178.319,5.786,148.523
C04324=1215.980,123.142,-50.370,-178.322,5.786,148.524
C04325=1215.984,122.893,-50.351,-178.325,5.784,148.524
C04326=1215.990,122.644,-50.332,-178.327,5.783,148.525
C04327=1215.994,122.395,-50.312,-178.330,5.782,148.525
C04328=1215.999,122.146,-50.292,-178.332,5.781,148.526
C04329=1216.004,121.897,-50.272,-178.335,5.780,148.526
C04330=1216.009,121.647,-50.253,-178.338,5.779,148.527
C04331=1216.013,121.398,-50.232,-178.340,5.778,148.527
C04332=1216.018,121.149,-50.213,-178.343,5.776,148.528
C04333=1216.023,120.900,-50.193,-178.345,5.775,148.528
C04334=1216.028,120.650,-50.174,-178.348,5.775,148.529
C04335=1216.033,120.401,-50.153,-178.350,5.773,148.529
C04336=1216.038,120.152,-50.134,-178.353,5.772,148.530
C04337=1216.043,119.903,-50.114,-178.356,5.771,148.530
C04338=1216.047,119.654,-50.095,-178.358,5.770,148.531
C04339=1216.052,119.405,-50.076,-178.360,5.769,148.532
C04340=1216.057,119.156,-50.056,-178.364,5.767,148.532
C04341=1216.061,118.906,-50.036,-178.366,5.767,148.533
C04342=1216.067,118.657,-50.017,-178.368,5.766,148.533
C04343=1216.071,118.408,-49.997,-178.371,5.764,148.534
C04344=1216.076,118.158,-49.977,-178.374,5.764,148.534
C04345=1216.081,117.910,-49.959,-178.376,5.763,148.535
C04346=1216.085,117.661,-49.938,-178.379,5.761,148.535
C04347=1216.090,117.411,-49.919,-178.381,5.760,148.536
C04348=1216.095,117.162,-49.899,-178.384,5.759,148.536
C04349=1216.100,116.913,-49.880,-178.386,5.758,148.537
C04350=1216.105,116.663,-49.860,-178.389,5.757,148.537
C04351=1216.109,116.415,-49.841,-178.392,5.755,148.538
C04352=1216.114,116.165,-49.822,-178.394,5.755,148.538
C04353=1216.119,115.916,-49.803,-178.396,5.754,148.539
C04354=1216.124,115.667,-49.783,-178.400,5.752,148.539
C04355=1216.128,115.417,-49.764,-178.402,5.752,148.540
C04356=1216.133,115.168,-49.744,-178.404,5.751,148.540
C04357=1216.138,114.919,-49.725,-178.408,5.749,148.541
C04358=1216.144,114.670,-49.706,-178.410,5.748,148.542
C04359=1216.148,114.420,-49.686,-178.412,5.748,148.542
C04360=1216.152,114.171,-49.667,-178.415,5.746,148.543
C04361=1216.158,113.922,-49.648,-178.418,5.745,148.543
C04362=1216.162,113.673,-49.628,-178.420,5.744,148.544
C04363=1216.167,113.424,-49.609,-178.423,5.743,148.544
C04364=1216.172,113.175,-49.590,-178.425,5.742,148.545
C04365=1216.177,112.925,-49.570,-178.428,5.742,148.545
C04366=1216.182,112.676,-49.551,-178.430,5.740,148.546
C04367=1216.186,112.427,-49.532,-178.433,5.739,148.546
C04368=1216.191,112.178,-49.512,-178.435,5.739,148.547
C04369=1216.196,111.928,-49.493,-178.438,5.737,148.547
C04370=1216.201,111.680,-49.474,-178.441,5.736,148.548
C04371=1216.205,111.430,-49.454,-178.443,5.735,148.548
C04372=1216.211,111.181,-49.436,-178.446,5.734,148.549
C04373=1216.215,110.932,-49.417,-178.448,5.733,148.549
C04374=1216.220,110.682,-49.397,-178.451,5.732,148.550
C04375=1216.225,110.433,-49.378,-178.454,5.730,148.550
C04376=1216.229,110.184,-49.359,-178.456,5.730,148.551
C04377=1216.234,109.935,-49.339,-178.459,5.729,148.552
C04378=1216.238,109.686,-49.320,-178.461,5.727,148.552
C04379=1216.244,109.436,-49.302,-178.464,5.727,148.553
C04380=1216.249,109.187,-49.282,-178.466,5.726,148.553
C04381=1216.253,108.938,-49.263,-178.469,5.724,148.554
C04382=1216.258,108.689,-49.244,-178.471,5.723,148.554
C04383=1216.263,108.440,-49.225,-178.474,5.723,148.555
C04384=1216.268,108.190,-49.206,-178.477,5.721,148.555
C04385=1216.273,107.941,-49.187,-178.479,5.721,148.556
C04386=1216.277,107.673,-49.166,-178.482,5.720,148.557
C04387=1216.283,107.404,-49.146,-178.485,5.718,148.557
C04388=1216.288,107.135,-49.125,-178.487,5.718,148.558
C04389=1216.294,106.867,-49.104,-178.491,5.716,148.558
C04390=1216.298,106.618,-49.086,-178.493,5.716,148.559
C04391=1216.303,106.369,-49.067,-178.495,5.715,148.559
C04392=1216.308,106.120,-49.048,-178.498,5.713,148.560
C04393=1216.313,105.870,-49.029,-178.501,5.712,148.560
C04394=1216.317,105.621,-49.010,-178.503,5.712,148.561
C04395=1216.322,105.372,-48.991,-178.506,5.710,148.562
C04396=1216.327,105.123,-48.973,-178.508,5.709,148.562
C04397=1216.332,104.873,-48.953,-178.511,5.709,148.563
C04398=1216.336,104.625,-48.934,-178.513,5.708,148.563
C04399=1216.342,104.375,-48.916,-178.516,5.706,148.564
C04400=1216.346,104.126,-48.897,-178.519,5.706,148.564
C04401=1216.352,103.876,-48.878,-178.521,5.705,148.565
C04402=1216.356,103.627,-48.859,-178.524,5.703,148.565
C04403=1216.361,103.378,-48.840,-178.526,5.702,148.566
C04404=1216.365,103.128,-48.822,-178.529,5.702,148.567
C04405=1216.371,102.879,-48.802,-178.532,5.701,148.567
C04406=1216.376,102.630,-48.784,-178.534,5.699,148.568
C04407=1216.380,102.381,-48.765,-178.537,5.699,148.568
C04408=1216.385,102.132,-48.747,-178.539,5.698,148.569
C04409=1216.389,101.882,-48.728,-178.542,5.696,148.569
C04410=1216.395,101.633,-48.708,-178.545,5.696,148.570
C04411=1216.400,101.384,-48.690,-178.547,5.695,148.570
C04412=1216.404,101.135,-48.671,-178.550,5.694,148.571
C04413=1216.409,100.886,-48.653,-178.552,5.692,148.571
C04414=1216.414,100.637,-48.634,-178.555,5.692,148.572
C04415=1216.419,100.387,-48.615,-178.558,5.691,148.573
C04416=1216.424,100.138,-48.596,-178.560,5.690,148.573
C04417=1216.429,99.888,-48.577,-178.563,5.689,148.574
C04418=1216.433,99.639,-48.559,-178.565,5.688,148.574
C04419=1216.438,99.390,-48.541,-178.568,5.687,148.575
C04420=1216.443,99.140,-48.522,-178.570,5.687,148.575
C04421=1216.448,98.892,-48.503,-178.573,5.685,148.576
C04422=1216.453,98.642,-48.485,-178.576,5.684,148.577
C04423=1216.457,98.393,-48.465,-178.578,5.683,148.577
C04424=1216.462,98.144,-48.447,-178.580,5.683,148.578
C04425=1216.467,97.894,-48.429,-178.584,5.681,148.578
C04426=1216.472,97.645,-48.410,-178.586,5.680,148.579
C04427=1216.477,97.396,-48.392,-178.588,5.680,148.579
C04428=1216.482,97.147,-48.374,-178.591,5.679,148.580
C04429=1216.487,96.897,-48.354,-178.594,5.678,148.580
C04430=1216.491,96.648,-48.336,-178.596,5.677,148.581
C04431=1216.496,96.399,-48.318,-178.598,5.676,148.581
C04432=1216.501,96.150,-48.300,-178.601,5.675,148.582
C04433=1216.506,95.900,-48.281,-178.604,5.674,148.583
C04434=1216.511,95.651,-48.263,-178.606,5.673,148.583
C04435=1216.516,95.402,-48.244,-178.609,5.672,148.584
C04436=1216.520,95.152,-48.226,-178.612,5.672,148.584
C04437=1216.525,94.903,-48.207,-178.614,5.670,148.585
C04438=1216.530,94.654,-48.188,-178.617,5.670,148.585
C04439=1216.535,94.405,-48.170,-178.619,5.669,148.586
C04440=1216.539,94.155,-48.152,-178.622,5.668,148.587
C04441=1216.545,93.906,-48.133,-178.624,5.667,148.587
C04442=1216.550,93.657,-48.115,-178.627,5.666,148.588
C04443=1216.554,93.408,-48.097,-178.630,5.665,148.588
C04444=1216.559,93.158,-48.078,-178.632,5.664,148.589
C04445=1216.564,92.909,-48.060,-178.634,5.663,148.589
C04446=1216.569,92.659,-48.042,-178.637,5.662,148.590
C04447=1216.574,92.411,-48.023,-178.640,5.661,148.591
C04448=1216.578,92.161,-48.005,-178.642,5.661,148.591
C04449=1216.583,91.912,-47.987,-178.645,5.660,148.592
C04450=1216.588,91.663,-47.969,-178.647,5.659,148.592
C04451=1216.593,91.413,-47.951,-178.650,5.658,148.593
C04452=1216.598,91.163,-47.932,-178.653,5.657,148.593
C04453=1216.603,90.915,-47.913,-178.655,5.656,148.594
C04454=1216.608,90.666,-47.895,-178.658,5.655,148.594
C04455=1216.612,90.416,-47.877,-178.661,5.654,148.595
C04456=1216.617,90.167,-47.859,-178.663,5.653,148.596
C04457=1216.622,89.917,-47.841,-178.665,5.653,148.596
C04458=1216.627,89.668,-47.823,-178.668,5.652,148.597
C04459=1216.632,89.419,-47.804,-178.670,5.651,148.597
C04460=1216.637,89.169,-47.786,-178.673,5.650,148.598
C04461=1216.642,88.920,-47.768,-178.676,5.649,148.599
C04462=1216.647,88.671,-47.750,-178.678,5.648,148.599
C04463=1216.651,88.421,-47.732,-178.681,5.647,148.600
C04464=1216.656,88.172,-47.714,-178.683,5.647,148.600
C04465=1216.661,87.923,-47.696,-178.686,5.645,148.601
C04466=1216.666,87.674,-47.677,-178.689,5.645,148.601
C04467=1216.671,87.425,-47.659,-178.691,5.644,148.602
C04468=1216.676,87.176,-47.642,-178.693,5.643,148.602
C04469=1216.680,86.926,-47.623,-178.696,5.642,148.603
C04470=1216.685,86.676,-47.606,-178.699,5.642,148.604
C04471=1216.690,86.427,-47.588,-178.701,5.640,148.604
C04472=1216.695,86.178,-47.570,-178.704,5.640,148.605
C04473=1216.700,85.929,-47.552,-178.707,5.639,148.605
C04474=1216.705,85.680,-47.534,-178.709,5.638,148.606
C04475=1216.710,85.430,-47.516,-178.711,5.637,148.607
C04476=1216.714,85.181,-47.498,-178.715,5.636,148.607
C04477=1216.719,84.931,-47.480,-178.717,5.635,148.608
C04478=1216.724,84.682,-47.462,-178.719,5.634,148.608
C04479=1216.729,84.433,-47.444,-178.722,5.634,148.609
C04480=1216.734,84.184,-47.426,-178.725,5.633,148.610
C04481=1216.739,83.935,-47.408,-178.727,5.632,148.610
C04482=1216.743,83.685,-47.390,-178.730,5.631,148.611
C04483=1216.749,83.436,-47.373,-178.733,5.630,148.611
C04484=1216.754,83.187,-47.355,-178.735,5.629,148.612
C04485=1216.758,82.937,-47.337,-178.737,5.629,148.612
C04486=1216.763,82.687,-47.318,-178.740,5.628,148.613
C04487=1216.768,82.438,-47.300,-178.742,5.627,148.613
C04488=1216.773,82.189,-47.282,-178.745,5.626,148.614
C04489=1216.778,81.939,-47.265,-178.748,5.625,148.615
C04490=1216.783,81.671,-47.246,-178.751,5.625,148.615
C04491=1216.788,81.403,-47.226,-178.753,5.624,148.616
C04492=1216.794,81.135,-47.207,-178.756,5.623,148.617
C04493=1216.799,80.866,-47.188,-178.758,5.622,148.617
C04494=1216.804,80.617,-47.170,-178.761,5.621,148.618
C04495=1216.809,80.368,-47.152,-178.764,5.621,148.618
C04496=1216.814,80.118,-47.135,-178.767,5.619,148.619
C04497=1216.818,79.869,-47.118,-178.769,5.618,148.620
C04498=1216.823,79.619,-47.099,-178.772,5.618,148.620
C04499=1216.828,79.370,-47.081,-178.774,5.617,148.621
C04500=1216.833,79.121,-47.064,-178.776,5.616,148.621
C04501=1216.838,78.871,-47.046,-178.779,5.616,148.622
C04502=1216.843,78.622,-47.028,-178.782,5.615,148.623
C04503=1216.848,78.372,-47.011,-178.784,5.613,148.623
C04504=1216.852,78.124,-46.994,-178.787,5.613,148.624
C04505=1216.857,77.874,-46.976,-178.790,5.612,148.624
C04506=1216.862,77.625,-46.958,-178.792,5.612,148.625
C04507=1216.867,77.375,-46.940,-178.794,5.611,148.625
C04508=1216.872,77.126,-46.922,-178.797,5.610,148.626
C04509=1216.876,76.877,-46.906,-178.800,5.610,148.627
C04510=1216.881,76.628,-46.888,-178.802,5.608,148.627
C04511=1216.886,76.378,-46.870,-178.805,5.607,148.628
C04512=1216.891,76.129,-46.853,-178.808,5.607,148.628
C04513=1216.896,75.879,-46.835,-178.810,5.606,148.629
C04514=1216.901,75.631,-46.818,-178.812,5.605,148.630
C04515=1216.906,75.381,-46.800,-178.815,5.605,148.630
C04516=1216.911,75.132,-46.782,-178.818,5.604,148.631
C04517=1216.916,74.882,-46.765,-178.820,5.603,148.632
C04518=1216.921,74.634,-46.748,-178.823,5.602,148.632
C04519=1216.926,74.384,-46.730,-178.826,5.601,148.633
C04520=1216.931,74.135,-46.712,-178.828,5.600,148.633
C04521=1216.936,73.885,-46.695,-178.830,5.600,148.634
C04522=1216.940,73.636,-46.678,-178.833,5.599,148.634
C04523=1216.945,73.386,-46.660,-178.836,5.598,148.635
C04524=1216.950,73.137,-46.642,-178.838,5.598,148.636
C04525=1216.955,72.888,-46.626,-178.840,5.597,148.636
C04526=1216.960,72.638,-46.608,-178.843,5.596,148.637
C04527=1216.965,72.389,-46.591,-178.846,5.595,148.637
C04528=1216.969,72.140,-46.573,-178.849,5.594,148.638
C04529=1216.974,71.890,-46.556,-178.851,5.593,148.639
C04530=1216.980,71.641,-46.538,-178.854,5.593,148.639
C04531=1216.984,71.392,-46.522,-178.856,5.592,148.640
C04532=1216.990,71.142,-46.504,-178.859,5.592,148.640
C04533=1216.994,70.893,-46.486,-178.861,5.591,148.641
C04534=1216.999,70.643,-46.470,-178.864,5.590,148.642
C04535=1217.004,70.394,-46.452,-178.866,5.590,148.642
C04536=1217.009,70.144,-46.434,-178.869,5.588,148.643
C04537=1217.014,69.895,-46.418,-178.872,5.587,148.643
C04538=1217.018,69.646,-46.400,-178.874,5.587,148.644
C04539=1217.024,69.397,-46.383,-178.877,5.586,148.645
C04540=1217.028,69.148,-46.366,-178.879,5.585,148.645
C04541=1217.034,68.898,-46.348,-178.882,5.585,148.646
C04542=1217.038,68.649,-46.332,-178.884,5.584,148.646
C04543=1217.043,68.399,-46.314,-178.887,5.584,148.647
C04544=1217.047,68.150,-46.297,-178.889,5.583,148.647
C04545=1217.053,67.900,-46.280,-178.892,5.582,148.648
C04546=1217.058,67.652,-46.262,-178.894,5.581,148.649
C04547=1217.063,67.402,-46.245,-178.898,5.580,148.649
C04548=1217.068,67.152,-46.228,-178.900,5.580,148.650
C04549=1217.072,66.903,-46.211,-178.902,5.579,148.651
C04550=1217.077,66.654,-46.194,-178.905,5.578,148.651
C04551=1217.082,66.404,-46.177,-178.908,5.577,148.652
C04552=1217.088,66.155,-46.160,-178.910,5.577,148.653
C04553=1217.092,65.906,-46.143,-178.912,5.576,148.653
C04554=1217.097,65.656,-46.125,-178.915,5.575,148.654
C04555=1217.101,65.407,-46.109,-178.918,5.575,148.654
C04556=1217.107,65.157,-46.091,-178.920,5.574,148.655
C04557=1217.112,64.908,-46.075,-178.922,5.573,148.655
C04558=1217.117,64.659,-46.057,-178.925,5.573,148.656
C04559=1217.121,64.410,-46.040,-178.928,5.572,148.657
C04560=1217.126,64.160,-46.023,-178.931,5.571,148.657
C04561=1217.131,63.910,-46.006,-178.933,5.570,148.658
C04562=1217.137,63.661,-45.990,-178.936,5.569,148.658
C04563=1217.141,63.412,-45.973,-178.938,5.569,148.659
C04564=1217.146,63.163,-45.955,-178.941,5.568,148.660
C04565=1217.151,62.913,-45.938,-178.943,5.568,148.660
C04566=1217.156,62.663,-45.921,-178.946,5.567,148.661
C04567=1217.161,62.415,-45.905,-178.948,5.566,148.662
C04568=1217.166,62.165,-45.887,-178.951,5.566,148.662
C04569=1217.171,61.915,-45.871,-178.954,5.565,148.663
C04570=1217.175,61.666,-45.854,-178.956,5.564,148.663
C04571=1217.181,61.417,-45.837,-178.958,5.564,148.664
C04572=1217.185,61.168,-45.820,-178.961,5.563,148.665
C04573=1217.190,60.918,-45.803,-178.964,5.562,148.665
C04574=1217.195,60.669,-45.786,-178.966,5.562,148.666
C04575=1217.201,60.420,-45.769,-178.968,5.561,148.666
C04576=1217.205,60.170,-45.752,-178.971,5.560,148.667
C04577=1217.210,59.921,-45.736,-178.974,5.559,148.668
C04578=1217.215,59.672,-45.719,-178.977,5.558,148.668
C04579=1217.220,59.422,-45.702,-178.979,5.557,148.669
C04580=1217.224,59.173,-45.685,-178.982,5.557,148.670
C04581=1217.230,58.923,-45.668,-178.984,5.556,148.670
C04582=1217.235,58.674,-45.652,-178.987,5.556,148.671
C04583=1217.239,58.424,-45.635,-178.990,5.555,148.672
C04584=1217.244,58.175,-45.618,-178.992,5.554,148.672
C04585=1217.249,57.926,-45.602,-178.994,5.554,148.673
C04586=1217.255,57.676,-45.584,-178.997,5.553,148.673
C04587=1217.259,57.427,-45.568,-179.000,5.553,148.674
C04588=1217.264,57.178,-45.551,-179.002,5.552,148.675
C04589=1217.269,56.928,-45.535,-179.004,5.551,148.675
C04590=1217.274,56.679,-45.517,-179.007,5.551,148.676
C04591=1217.279,56.429,-45.502,-179.010,5.550,148.676
C04592=1217.284,56.180,-45.485,-179.012,5.549,148.677
C04593=1217.289,55.930,-45.468,-179.015,5.549,148.678
C04594=1217.294,55.662,-45.450,-179.017,5.548,148.678
C04595=1217.299,55.393,-45.432,-179.020,5.548,148.679
C04596=1217.305,55.125,-45.414,-179.023,5.546,148.680
C04597=1217.310,54.857,-45.397,-179.026,5.546,148.680
C04598=1217.315,54.607,-45.380,-179.028,5.545,148.681
C04599=1217.320,54.358,-45.363,-179.031,5.544,148.682
C04600=1217.325,54.109,-45.346,-179.033,5.544,148.682
C04601=1217.330,53.859,-45.331,-179.036,5.543,148.683
C04602=1217.334,53.609,-45.314,-179.039,5.543,148.684
C04603=1217.340,53.360,-45.298,-179.041,5.542,148.684
C04604=1217.345,53.111,-45.280,-179.043,5.541,148.685
C04605=1217.350,52.862,-45.264,-179.046,5.541,148.685
C04606=1217.355,52.612,-45.248,-179.049,5.540,148.686
C04607=1217.359,52.362,-45.231,-179.051,5.540,148.687
C04608=1217.365,52.113,-45.214,-179.053,5.539,148.687
C04609=1217.369,51.864,-45.198,-179.056,5.538,148.688
C04610=1217.374,51.615,-45.181,-179.059,5.537,148.688
C04611=1217.379,51.365,-45.166,-179.061,5.537,148.689
C04612=1217.384,51.115,-45.149,-179.064,5.536,148.690
C04613=1217.389,50.866,-45.133,-179.067,5.536,148.690
C04614=1217.394,50.616,-45.116,-179.069,5.535,148.691
C04615=1217.399,50.367,-45.100,-179.071,5.534,148.692
C04616=1217.404,50.118,-45.083,-179.074,5.534,148.692
C04617=1217.408,49.868,-45.066,-179.077,5.533,148.693
C04618=1217.414,49.619,-45.051,-179.079,5.533,148.694
C04619=1217.418,49.369,-45.034,-179.082,5.532,148.694
C04620=1217.423,49.121,-45.018,-179.084,5.531,148.695
C04621=1217.429,48.870,-45.001,-179.087,5.531,148.695
C04622=1217.434,48.621,-44.985,-179.089,5.530,148.696
C04623=1217.438,48.372,-44.968,-179.092,5.530,148.697
C04624=1217.444,48.123,-44.953,-179.095,5.529,148.697
C04625=1217.448,47.873,-44.936,-179.097,5.528,148.698
C04626=1217.454,47.624,-44.920,-179.099,5.528,148.698
C04627=1217.458,47.374,-44.904,-179.102,5.527,148.699
C04628=1217.463,47.125,-44.887,-179.105,5.526,148.700
C04629=1217.468,46.875,-44.872,-179.107,5.526,148.700
C04630=1217.472,46.626,-44.855,-179.110,5.525,148.701
C04631=1217.478,46.376,-44.839,-179.112,5.524,148.702
C04632=1217.482,46.127,-44.823,-179.115,5.524,148.702
C04633=1217.487,45.878,-44.806,-179.117,5.523,148.703
C04634=1217.493,45.628,-44.790,-179.120,5.523,148.704
C04635=1217.498,45.379,-44.773,-179.123,5.522,148.704
C04636=1217.503,45.129,-44.757,-179.125,5.522,148.705
C04637=1217.508,44.880,-44.741,-179.128,5.521,148.705
C04638=1217.513,44.630,-44.725,-179.130,5.520,148.706
C04639=1217.518,44.381,-44.709,-179.133,5.520,148.707
C04640=1217.523,44.131,-44.693,-179.135,5.519,148.707
C04641=1217.528,43.882,-44.677,-179.138,5.519,148.708
C04642=1217.533,43.633,-44.661,-179.141,5.518,148.709
C04643=1217.537,43.383,-44.644,-179.143,5.517,148.709
C04644=1217.543,43.134,-44.629,-179.146,5.517,148.710
C04645=1217.547,42.885,-44.612,-179.148,5.517,148.711
C04646=1217.553,42.635,-44.597,-179.150,5.516,148.711
C04647=1217.557,42.386,-44.580,-179.153,5.516,148.712
C04648=1217.563,42.136,-44.564,-179.155,5.515,148.713
C04649=1217.567,41.886,-44.548,-179.158,5.514,148.713
C04650=1217.572,41.638,-44.533,-179.160,5.514,148.714
C04651=1217.577,41.388,-44.517,-179.163,5.513,148.714
C04652=1217.582,41.139,-44.500,-179.166,5.513,148.715
C04653=1217.587,40.889,-44.485,-179.168,5.512,148.716
C04654=1217.592,40.639,-44.469,-179.171,5.511,148.716
C04655=1217.597,40.390,-44.453,-179.173,5.511,148.717
C04656=1217.602,40.140,-44.437,-179.176,5.510,148.717
C04657=1217.607,39.891,-44.421,-179.178,5.509,148.718
C04658=1217.612,39.642,-44.405,-179.181,5.509,148.719
C04659=1217.617,39.392,-44.389,-179.184,5.508,148.719
C04660=1217.622,39.143,-44.372,-179.186,5.508,148.720
C04661=1217.627,38.893,-44.356,-179.189,5.507,148.721
C04662=1217.631,38.644,-44.342,-179.191,5.507,148.721
C04663=1217.637,38.395,-44.326,-179.194,5.506,148.722
C04664=1217.641,38.145,-44.309,-179.196,5.505,148.723
C04665=1217.647,37.896,-44.294,-179.199,5.505,148.723
C04666=1217.651,37.646,-44.278,-179.201,5.505,148.724
C04667=1217.657,37.397,-44.261,-179.204,5.504,148.725
C04668=1217.662,37.148,-44.246,-179.206,5.504,148.725
C04669=1217.667,36.897,-44.230,-179.209,5.503,148.726
C04670=1217.671,36.648,-44.215,-179.211,5.502,148.726
C04671=1217.676,36.400,-44.199,-179.214,5.502,148.727
C04672=1217.681,36.149,-44.183,-179.216,5.501,148.728
C04673=1217.687,35.900,-44.167,-179.219,5.501,148.728
C04674=1217.692,35.651,-44.151,-179.222,5.500,148.729
C04675=1217.696,35.401,-44.136,-179.224,5.500,148.730
C04676=1217.701,35.152,-44.120,-179.227,5.499,148.730
C04677=1217.707,34.903,-44.104,-179.229,5.498,148.731
C04678=1217.711,34.653,-44.088,-179.232,5.498,148.732
C04679=1217.717,34.403,-44.073,-179.234,5.497,148.732
C04680=1217.721,34.154,-44.058,-179.237,5.497,148.733
C04681=1217.726,33.905,-44.041,-179.239,5.497,148.734
C04682=1217.731,33.655,-44.025,-179.242,5.496,148.734
C04683=1217.737,33.406,-44.010,-179.244,5.496,148.735
C04684=1217.741,33.156,-43.994,-179.247,5.495,148.736
C04685=1217.746,32.907,-43.979,-179.249,5.494,148.736
C04686=1217.751,32.657,-43.963,-179.252,5.494,148.737
C04687=1217.756,32.407,-43.947,-179.254,5.493,148.737
C04688=1217.761,32.158,-43.932,-179.257,5.493,148.738
C04689=1217.766,31.909,-43.916,-179.260,5.492,148.739
C04690=1217.771,31.660,-43.900,-179.262,5.492,148.740
C04691=1217.776,31.410,-43.884,-179.265,5.491,148.740
C04692=1217.781,31.161,-43.869,-179.268,5.491,148.741
C04693=1217.786,30.911,-43.854,-179.269,5.491,148.741
C04694=1217.791,30.661,-43.838,-179.272,5.490,148.742
C04695=1217.796,30.412,-43.823,-179.274,5.489,148.743
C04696=1217.801,30.163,-43.807,-179.277,5.489,148.743
C04697=1217.806,29.913,-43.792,-179.280,5.488,148.744
C04698=1217.811,29.644,-43.775,-179.282,5.488,148.745
C04699=1217.816,29.375,-43.759,-179.285,5.487,148.745
C04700=1217.822,29.107,-43.742,-179.288,5.487,148.746
C04701=1217.828,28.838,-43.725,-179.290,5.486,148.747
C04702=1217.832,28.589,-43.710,-179.293,5.486,148.747
C04703=1217.838,28.340,-43.694,-179.296,5.485,148.748
C04704=1217.842,28.090,-43.679,-179.298,5.485,148.749
C04705=1217.847,27.841,-43.663,-179.301,5.484,148.749
C04706=1217.852,27.591,-43.648,-179.304,5.484,148.750
C04707=1217.857,27.342,-43.633,-179.306,5.483,148.751
C04708=1217.862,27.093,-43.617,-179.309,5.483,148.751
C04709=1217.868,26.842,-43.602,-179.310,5.482,148.752
C04710=1217.872,26.593,-43.587,-179.313,5.482,148.753
C04711=1217.878,26.343,-43.571,-179.316,5.481,148.753
C04712=1217.882,26.094,-43.556,-179.318,5.481,148.754
C04713=1217.887,25.844,-43.540,-179.321,5.480,148.755
C04714=1217.892,25.595,-43.525,-179.324,5.480,148.755
C04715=1217.897,25.346,-43.510,-179.326,5.479,148.756
C04716=1217.902,25.096,-43.494,-179.329,5.479,148.757
C04717=1217.907,24.847,-43.479,-179.332,5.478,148.757
C04718=1217.913,24.597,-43.464,-179.333,5.478,148.758
C04719=1217.917,24.347,-43.449,-179.336,5.478,148.758
C04720=1217.922,24.098,-43.433,-179.338,5.477,148.759
C04721=1217.927,23.849,-43.418,-179.341,5.476,148.760
C04722=1217.932,23.600,-43.403,-179.344,5.476,148.761
C04723=1217.937,23.350,-43.388,-179.346,5.475,148.761
C04724=1217.943,23.100,-43.373,-179.349,5.475,148.762
C04725=1217.947,22.851,-43.357,-179.352,5.474,148.763
C04726=1217.952,22.601,-43.342,-179.354,5.475,148.763
C04727=1217.957,22.352,-43.327,-179.356,5.474,148.764
C04728=1217.962,22.103,-43.311,-179.359,5.473,148.764
C04729=1217.967,21.853,-43.297,-179.361,5.473,148.765
C04730=1217.972,21.604,-43.281,-179.364,5.472,148.766
C04731=1217.976,21.354,-43.266,-179.367,5.472,148.766
C04732=1217.982,21.104,-43.250,-179.369,5.471,148.767
C04733=1217.987,20.855,-43.236,-179.372,5.471,148.768
C04734=1217.992,20.605,-43.221,-179.374,5.471,148.768
C04735=1217.997,20.356,-43.206,-179.377,5.470,148.769
C04736=1218.003,20.106,-43.191,-179.379,5.470,148.770
C04737=1218.007,19.857,-43.176,-179.382,5.469,148.771
C04738=1218.013,19.608,-43.160,-179.384,5.468,148.771
C04739=1218.017,19.359,-43.145,-179.387,5.468,148.772
C04740=1218.022,19.108,-43.130,-179.389,5.467,148.772
C04741=1218.027,18.859,-43.115,-179.391,5.468,148.773
C04742=1218.032,18.610,-43.100,-179.394,5.467,148.774
C04743=1218.037,18.360,-43.085,-179.397,5.466,148.774
C04744=1218.042,18.111,-43.070,-179.399,5.466,148.775
C04745=1218.048,17.861,-43.055,-179.402,5.465,148.776
C04746=1218.052,17.612,-43.040,-179.405,5.465,148.776
C04747=1218.057,17.362,-43.025,-179.407,5.464,148.777
C04748=1218.063,17.112,-43.010,-179.409,5.464,148.778
C04749=1218.067,16.863,-42.995,-179.411,5.464,148.778
C04750=1218.073,16.613,-42.980,-179.414,5.463,148.779
C04751=1218.078,16.364,-42.965,-179.417,5.463,148.780
C04752=1218.082,16.115,-42.950,-179.419,5.462,148.780
C04753=1218.087,15.864,-42.935,-179.422,5.462,148.781
C04754=1218.092,15.615,-42.920,-179.424,5.462,148.782
C04755=1218.097,15.366,-42.906,-179.427,5.461,148.782
C04756=1218.102,15.116,-42.890,-179.429,5.461,148.783
C04757=1218.107,14.866,-42.876,-179.432,5.460,148.784
C04758=1218.112,14.617,-42.861,-179.435,5.460,148.784
C04759=1218.118,14.367,-42.846,-179.437,5.459,148.785
C04760=1218.122,14.118,-42.831,-179.439,5.459,148.786
C04761=1218.127,13.869,-42.816,-179.442,5.459,148.786
C04762=1218.133,13.619,-42.801,-179.444,5.458,148.787
C04763=1218.137,13.370,-42.786,-179.447,5.458,148.788
C04764=1218.142,13.120,-42.772,-179.450,5.457,148.788
C04765=1218.147,12.871,-42.758,-179.452,5.457,148.789
C04766=1218.153,12.621,-42.742,-179.454,5.457,148.790
C04767=1218.158,12.372,-42.728,-179.457,5.456,148.790
C04768=1218.162,12.122,-42.713,-179.460,5.456,148.791
C04769=1218.168,11.872,-42.698,-179.462,5.455,148.792
C04770=1218.173,11.623,-42.683,-179.465,5.455,148.792
C04771=1218.177,11.374,-42.669,-179.468,5.454,148.793
C04772=1218.182,11.125,-42.654,-179.469,5.454,148.794
C04773=1218.188,10.875,-42.639,-179.472,5.454,148.794
C04774=1218.193,10.625,-42.625,-179.474,5.453,148.795
C04775=1218.197,10.376,-42.610,-179.477,5.453,148.796
C04776=1218.202,10.126,-42.595,-179.480,5.452,148.796
C04777=1218.207,9.877,-42.580,-179.482,5.452,148.797
C04778=1218.213,9.627,-42.566,-179.484,5.452,148.798
C04779=1218.218,9.377,-42.551,-179.487,5.451,148.798
C04780=1218.222,9.128,-42.536,-179.490,5.451,148.799
C04781=1218.228,8.879,-42.522,-179.492,5.450,148.800
C04782=1218.234,8.629,-42.507,-179.495,5.450,148.800
C04783=1218.238,8.380,-42.492,-179.497,5.450,148.801
C04784=1218.243,8.130,-42.478,-179.500,5.450,148.802
C04785=1218.248,7.881,-42.464,-179.502,5.449,148.802
C04786=1218.253,7.631,-42.449,-179.505,5.448,148.803
C04787=1218.258,7.382,-42.435,-179.507,5.448,148.804
C04788=1218.263,7.132,-42.420,-179.509,5.448,148.804
C04789=1218.268,6.882,-42.406,-179.512,5.447,148.805
C04790=1218.273,6.633,-42.391,-179.515,5.447,148.806
C04791=1218.278,6.383,-42.376,-179.517,5.446,148.806
C04792=1218.283,6.133,-42.362,-179.520,5.446,148.807
C04793=1218.288,5.884,-42.347,-179.523,5.445,148.808
C04794=1218.293,5.635,-42.333,-179.525,5.446,148.808
C04795=1218.299,5.385,-42.318,-179.527,5.445,148.809
C04796=1218.304,5.136,-42.304,-179.530,5.445,148.810
C04797=1218.309,4.886,-42.290,-179.533,5.444,148.810
C04798=1218.313,4.637,-42.275,-179.535,5.444,148.811
C04799=1218.318,4.387,-42.260,-179.537,5.444,148.812
C04800=1218.323,4.137,-42.246,-179.540,5.443,148.813
C04801=1218.328,3.888,-42.232,-179.542,5.442,148.813
C04802=1218.333,3.619,-42.216,-179.545,5.442,148.814
C04803=1218.339,3.351,-42.201,-179.548,5.442,148.815
C04804=1218.345,3.081,-42.185,-179.551,5.441,148.815
C04805=1218.350,2.812,-42.169,-179.553,5.441,148.816
C04806=1218.355,2.563,-42.155,-179.555,5.441,148.817
C04807=1218.360,2.313,-42.141,-179.558,5.441,148.817
C04808=1218.365,2.063,-42.127,-179.561,5.440,148.818
C04809=1218.370,1.813,-42.112,-179.563,5.440,148.819
C04810=1218.375,1.565,-42.098,-179.566,5.439,148.819
C04811=1218.380,1.315,-42.083,-179.568,5.439,148.820
C04812=1218.385,1.066,-42.069,-179.571,5.439,148.821
C04813=1218.390,0.816,-42.055,-179.573,5.438,148.821
C04814=1218.395,0.566,-42.041,-179.576,5.438,148.822
C04815=1218.400,0.317,-42.026,-179.578,5.438,148.823
C04816=1218.406,0.068,-42.012,-179.580,5.437,148.823
C04817=1218.411,-0.182,-41.998,-179.583,5.437,148.824
C04818=1218.416,-0.432,-41.984,-179.585,5.436,148.825
C04819=1218.421,-0.682,-41.970,-179.588,5.436,148.825
C04820=1218.426,-0.931,-41.955,-179.590,5.436,148.826
C04821=1218.431,-1.180,-41.941,-179.593,5.435,148.827
C04822=1218.436,-1.430,-41.927,-179.596,5.435,148.827
C04823=1218.441,-1.680,-41.913,-179.598,5.434,148.828
C04824=1218.446,-1.929,-41.899,-179.600,5.435,148.829
C04825=1218.451,-2.179,-41.884,-179.603,5.434,148.830
C04826=1218.457,-2.428,-41.870,-179.606,5.434,148.830
C04827=1218.462,-2.678,-41.856,-179.608,5.433,148.831
C04828=1218.466,-2.928,-41.842,-179.611,5.433,148.832
C04829=1218.471,-3.177,-41.828,-179.613,5.433,148.832
C04830=1218.477,-3.426,-41.814,-179.616,5.432,148.833
C04831=1218.482,-3.676,-41.799,-179.618,5.432,148.834
C04832=1218.486,-3.925,-41.786,-179.621,5.431,148.834
C04833=1218.491,-4.175,-41.771,-179.622,5.431,148.835
C04834=1218.496,-4.425,-41.757,-179.625,5.431,148.835
C04835=1218.502,-4.674,-41.743,-179.628,5.430,148.836
C04836=1218.507,-4.924,-41.729,-179.630,5.430,148.837
C04837=1218.512,-5.173,-41.715,-179.633,5.430,148.838
C04838=1218.517,-5.422,-41.701,-179.635,5.430,148.838
C04839=1218.522,-5.672,-41.686,-179.638,5.429,148.839
C04840=1218.527,-5.922,-41.673,-179.640,5.429,148.840
C04841=1218.532,-6.172,-41.659,-179.643,5.429,148.840
C04842=1218.537,-6.421,-41.645,-179.645,5.428,148.841
C04843=1218.542,-6.670,-41.631,-179.648,5.428,148.842
C04844=1218.547,-6.920,-41.617,-179.651,5.427,148.842
C04845=1218.552,-7.170,-41.603,-179.653,5.428,148.843
C04846=1218.557,-7.419,-41.589,-179.655,5.427,148.844
C04847=1218.562,-7.669,-41.576,-179.658,5.427,148.844
C04848=1218.567,-7.919,-41.561,-179.661,5.426,148.845
C04849=1218.573,-8.168,-41.547,-179.663,5.426,148.846
C04850=1218.577,-8.417,-41.533,-179.665,5.426,148.847
C04851=1218.582,-8.667,-41.519,-179.668,5.425,148.847
C04852=1218.587,-8.917,-41.506,-179.671,5.425,148.848
C04853=1218.593,-9.166,-41.492,-179.672,5.425,148.848
C04854=1218.597,-9.416,-41.478,-179.675,5.424,148.849
C04855=1218.602,-9.665,-41.463,-179.678,5.424,148.850
C04856=1218.608,-9.914,-41.450,-179.680,5.423,148.850
C04857=1218.612,-10.165,-41.437,-179.682,5.424,148.851
C04858=1218.617,-10.414,-41.422,-179.685,5.423,148.852
C04859=1218.623,-10.663,-41.408,-179.688,5.423,148.853
C04860=1218.628,-10.914,-41.395,-179.690,5.422,148.853
C04861=1218.632,-11.163,-41.381,-179.692,5.422,148.854
C04862=1218.638,-11.412,-41.367,-179.695,5.422,148.855
C04863=1218.643,-11.662,-41.353,-179.698,5.421,148.855
C04864=1218.648,-11.912,-41.339,-179.700,5.421,148.856
C04865=1218.653,-12.161,-41.326,-179.702,5.421,148.857
C04866=1218.658,-12.410,-41.312,-179.705,5.421,148.857
C04867=1218.664,-12.660,-41.299,-179.708,5.420,148.858
C04868=1218.669,-12.910,-41.284,-179.710,5.421,148.859
C04869=1218.673,-13.159,-41.271,-179.712,5.420,148.859
C04870=1218.679,-13.409,-41.257,-179.715,5.420,148.860
C04871=1218.684,-13.658,-41.243,-179.718,5.419,148.861
C04872=1218.688,-13.908,-41.229,-179.720,5.419,148.862
C04873=1218.694,-14.158,-41.216,-179.722,5.419,148.862
C04874=1218.699,-14.407,-41.202,-179.725,5.418,148.863
C04875=1218.704,-14.657,-41.189,-179.728,5.418,148.864
C04876=1218.709,-14.906,-41.175,-179.729,5.418,148.864
C04877=1218.714,-15.156,-41.161,-179.732,5.417,148.865
C04878=1218.719,-15.405,-41.148,-179.735,5.417,148.865
C04879=1218.724,-15.655,-41.134,-179.737,5.417,148.866
C04880=1218.730,-15.905,-41.121,-179.739,5.417,148.867
C04881=1218.734,-16.154,-41.107,-179.742,5.416,148.868
C04882=1218.739,-16.404,-41.093,-179.745,5.416,148.868
C04883=1218.745,-16.653,-41.080,-179.747,5.416,148.869
C04884=1218.749,-16.903,-41.066,-179.749,5.415,148.870
C04885=1218.755,-17.152,-41.053,-179.752,5.415,148.870
C04886=1218.760,-17.402,-41.038,-179.754,5.415,148.871
C04887=1218.765,-17.651,-41.026,-179.757,5.415,148.872
C04888=1218.770,-17.901,-41.012,-179.759,5.414,148.872
C04889=1218.775,-18.151,-40.999,-179.762,5.414,148.873
C04890=1218.780,-18.400,-40.985,-179.764,5.414,148.874
C04891=1218.785,-18.650,-40.971,-179.767,5.414,148.874
C04892=1218.790,-18.899,-40.958,-179.770,5.413,148.875
C04893=1218.795,-19.150,-40.944,-179.772,5.413,148.876
C04894=1218.800,-19.398,-40.931,-179.774,5.413,148.877
C04895=1218.806,-19.649,-40.917,-179.777,5.412,148.877
C04896=1218.811,-19.898,-40.903,-179.780,5.412,148.878
C04897=1218.816,-20.148,-40.891,-179.782,5.412,148.879
C04898=1218.821,-20.397,-40.877,-179.784,5.412,148.879
C04899=1218.826,-20.647,-40.864,-179.787,5.411,148.880
C04900=1218.832,-20.896,-40.850,-179.789,5.412,148.881
C04901=1218.836,-21.146,-40.837,-179.792,5.411,148.881
C04902=1218.842,-21.395,-40.824,-179.794,5.410,148.882
C04903=1218.846,-21.645,-40.810,-179.797,5.410,148.883
C04904=1218.852,-21.894,-40.797,-179.799,5.410,148.883
C04905=1218.856,-22.144,-40.784,-179.801,5.409,148.884
C04906=1218.862,-22.414,-40.769,-179.804,5.409,148.885
C04907=1218.868,-22.683,-40.755,-179.807,5.409,148.886
C04908=1218.873,-22.952,-40.740,-179.809,5.409,148.886
C04909=1218.878,-23.222,-40.725,-179.812,5.409,148.887
C04910=1218.884,-23.471,-40.712,-179.815,5.408,148.888
C04911=1218.889,-23.721,-40.699,-179.817,5.408,148.888
C04912=1218.894,-23.970,-40.685,-179.819,5.408,148.889
C04913=1218.899,-24.220,-40.672,-179.822,5.408,148.890
C04914=1218.904,-24.470,-40.660,-179.825,5.407,148.890
C04915=1218.909,-24.719,-40.646,-179.827,5.407,148.891
C04916=1218.914,-24.969,-40.633,-179.829,5.407,148.892
C04917=1218.919,-25.219,-40.619,-179.832,5.406,148.893
C04918=1218.924,-25.468,-40.607,-179.834,5.407,148.893
C04919=1218.930,-25.717,-40.593,-179.837,5.406,148.894
C04920=1218.934,-25.967,-40.580,-179.839,5.406,148.895
C04921=1218.940,-26.217,-40.567,-179.841,5.406,148.895
C04922=1218.944,-26.466,-40.553,-179.844,5.406,148.896
C04923=1218.949,-26.716,-40.540,-179.847,5.405,148.897
C04924=1218.955,-26.966,-40.527,-179.849,5.405,148.897
C04925=1218.960,-27.215,-40.514,-179.852,5.405,148.898
C04926=1218.965,-27.466,-40.501,-179.854,5.404,148.899
C04927=1218.970,-27.714,-40.487,-179.857,5.404,148.900
C04928=1218.975,-27.964,-40.475,-179.858,5.404,148.900
C04929=1218.980,-28.214,-40.461,-179.861,5.403,148.901
C04930=1218.985,-28.463,-40.449,-179.864,5.403,148.901
C04931=1218.991,-28.714,-40.435,-179.866,5.403,148.902
C04932=1218.996,-28.962,-40.422,-179.868,5.403,148.903
C04933=1219.001,-29.212,-40.409,-179.871,5.402,148.904
C04934=1219.006,-29.462,-40.396,-179.873,5.403,148.904
C04935=1219.011,-29.711,-40.383,-179.876,5.402,148.905
C04936=1219.016,-29.961,-40.370,-179.879,5.402,148.906
C04937=1219.021,-30.211,-40.357,-179.881,5.402,148.906
C04938=1219.026,-30.460,-40.343,-179.883,5.401,148.907
C04939=1219.031,-30.710,-40.331,-179.886,5.401,148.908
C04940=1219.037,-30.959,-40.317,-179.888,5.401,148.908
C04941=1219.042,-31.209,-40.305,-179.891,5.401,148.909
C04942=1219.046,-31.459,-40.292,-179.893,5.400,148.910
C04943=1219.052,-31.708,-40.279,-179.895,5.401,148.910
C04944=1219.057,-31.958,-40.266,-179.898,5.400,148.911
C04945=1219.062,-32.208,-40.253,-179.901,5.400,148.912
C04946=1219.068,-32.457,-40.240,-179.903,5.400,148.913
C04947=1219.072,-32.707,-40.227,-179.906,5.399,148.913
C04948=1219.077,-32.956,-40.214,-179.908,5.399,148.914
C04949=1219.082,-33.205,-40.201,-179.910,5.399,148.915
C04950=1219.087,-33.456,-40.187,-179.913,5.399,148.915
C04951=1219.092,-33.705,-40.175,-179.916,5.398,148.916
C04952=1219.098,-33.954,-40.162,-179.918,5.399,148.917
C04953=1219.102,-34.204,-40.149,-179.920,5.398,148.917
C04954=1219.108,-34.454,-40.136,-179.923,5.398,148.918
C04955=1219.113,-34.703,-40.123,-179.925,5.398,148.919
C04956=1219.118,-34.953,-40.110,-179.928,5.397,148.920
C04957=1219.123,-35.202,-40.098,-179.930,5.397,148.920
C04958=1219.129,-35.452,-40.085,-179.932,5.397,148.921
C04959=1219.133,-35.702,-40.072,-179.935,5.396,148.921
C04960=1219.138,-35.951,-40.059,-179.937,5.396,148.922
C04961=1219.143,-36.201,-40.046,-179.939,5.396,148.923
C04962=1219.149,-36.450,-40.033,-179.942,5.396,148.924
C04963=1219.154,-36.700,-40.020,-179.944,5.396,148.924
C04964=1219.159,-36.950,-40.008,-179.947,5.396,148.925
C04965=1219.164,-37.200,-39.996,-179.949,5.395,148.926
C04966=1219.169,-37.450,-39.983,-179.952,5.395,148.926
C04967=1219.175,-37.699,-39.970,-179.954,5.395,148.927
C04968=1219.180,-37.949,-39.957,-179.957,5.395,148.928
C04969=1219.185,-38.198,-39.944,-179.959,5.395,148.928
C04970=1219.189,-38.448,-39.931,-179.962,5.394,148.929
C04971=1219.195,-38.697,-39.919,-179.964,5.394,148.930
C04972=1219.200,-38.947,-39.906,-179.966,5.394,148.931
C04973=1219.206,-39.196,-39.893,-179.969,5.394,148.931
C04974=1219.210,-39.447,-39.881,-179.972,5.393,148.932
C04975=1219.216,-39.696,-39.868,-179.974,5.394,148.933
C04976=1219.221,-39.945,-39.856,-179.976,5.393,148.933
C04977=1219.226,-40.195,-39.843,-179.979,5.393,148.934
C04978=1219.230,-40.445,-39.830,-179.981,5.393,148.935
C04979=1219.235,-40.694,-39.817,-179.984,5.392,148.935
C04980=1219.242,-40.944,-39.805,-179.986,5.393,148.936
C04981=1219.247,-41.194,-39.792,-179.989,5.392,148.937
C04982=1219.251,-41.444,-39.779,-179.991,5.392,148.938
C04983=1219.256,-41.693,-39.767,-179.993,5.392,148.938
C04984=1219.261,-41.942,-39.754,-179.996,5.392,148.939
C04985=1219.267,-42.192,-39.742,-179.999,5.391,148.940
C04986=1219.271,-42.442,-39.729,179.999,5.392,148.940
C04987=1219.277,-42.692,-39.717,179.997,5.391,148.941
C04988=1219.282,-42.941,-39.704,179.995,5.391,148.942
C04989=1219.287,-43.190,-39.692,179.992,5.391,148.942
C04990=1219.292,-43.440,-39.680,179.990,5.390,148.943
C04991=1219.297,-43.690,-39.667,179.988,5.390,148.944
C04992=1219.303,-43.940,-39.653,179.985,5.390,148.944
C04993=1219.308,-44.189,-39.641,179.982,5.389,148.945
C04994=1219.313,-44.439,-39.629,179.980,5.390,148.946
C04995=1219.318,-44.688,-39.616,179.977,5.389,148.946
C04996=1219.323,-44.938,-39.604,179.975,5.390,148.947
C04997=1219.328,-45.188,-39.592,179.973,5.389,148.948
C04998=1219.333,-45.438,-39.579,179.970,5.389,148.949
C04999=1219.338,-45.687,-39.566,179.968,5.389,148.949
C05000=1219.344,-45.937,-39.554,179.965,5.389,148.950
C05001=1219.349,-46.186,-39.542,179.963,5.388,148.951
C05002=1219.354,-46.436,-39.529,179.961,5.388,148.951
C05003=1219.359,-46.686,-39.517,179.958,5.388,148.952
C05004=1219.364,-46.936,-39.504,179.956,5.388,148.953
C05005=1219.369,-47.185,-39.492,179.953,5.388,148.953
C05006=1219.375,-47.435,-39.480,179.951,5.387,148.954
C05007=1219.380,-47.684,-39.467,179.948,5.388,148.955
C05008=1219.385,-47.933,-39.455,179.946,5.387,148.956
C05009=1219.390,-48.183,-39.443,179.943,5.387,148.956
C05010=1219.395,-48.453,-39.429,179.941,5.387,148.957
C05011=1219.401,-48.723,-39.416,179.938,5.387,148.958
C05012=1219.406,-48.992,-39.403,179.936,5.386,148.958
C05013=1219.412,-49.263,-39.389,179.934,5.386,148.959
C05014=1219.417,-49.512,-39.377,179.931,5.386,148.960
C05015=1219.423,-49.762,-39.365,179.928,5.385,148.960
C05016=1219.427,-50.011,-39.353,179.926,5.386,148.961
C05017=1219.433,-50.261,-39.341,179.924,5.385,148.962
C05018=1219.437,-50.511,-39.328,179.921,5.385,148.963
C05019=1219.443,-50.761,-39.316,179.919,5.385,148.963
C05020=1219.448,-51.011,-39.303,179.916,5.385,148.964
C05021=1219.453,-51.261,-39.292,179.914,5.385,148.965
C05022=1219.458,-51.510,-39.279,179.911,5.385,148.965
C05023=1219.464,-51.760,-39.267,179.909,5.384,148.966
C05024=1219.469,-52.009,-39.255,179.907,5.384,148.967
C05025=1219.474,-52.259,-39.243,179.904,5.384,148.968
C05026=1219.479,-52.508,-39.231,179.902,5.384,148.968
C05027=1219.484,-52.758,-39.219,179.899,5.384,148.969
C05028=1219.489,-53.007,-39.206,179.896,5.383,148.970
C05029=1219.494,-53.258,-39.194,179.894,5.384,148.970
C05030=1219.499,-53.507,-39.181,179.892,5.383,148.971
C05031=1219.505,-53.757,-39.169,179.890,5.384,148.972
C05032=1219.509,-54.006,-39.157,179.887,5.383,148.972
C05033=1219.514,-54.256,-39.146,179.884,5.383,148.973
C05034=1219.520,-54.505,-39.133,179.882,5.383,148.974
C05035=1219.525,-54.755,-39.121,179.880,5.383,148.975
C05036=1219.530,-55.005,-39.109,179.877,5.383,148.975
C05037=1219.536,-55.255,-39.097,179.875,5.382,148.976
C05038=1219.540,-55.504,-39.085,179.873,5.382,148.976
C05039=1219.545,-55.754,-39.073,179.871,5.382,148.977
C05040=1219.551,-56.004,-39.061,179.868,5.381,148.978
C05041=1219.556,-56.253,-39.049,179.866,5.382,148.979
C05042=1219.561,-56.503,-39.036,179.863,5.381,148.979
C05043=1219.566,-56.752,-39.025,179.861,5.382,148.980
C05044=1219.571,-57.002,-39.012,179.858,5.381,148.981
C05045=1219.577,-57.252,-39.001,179.856,5.381,148.981
C05046=1219.582,-57.502,-38.989,179.854,5.381,148.982
C05047=1219.586,-57.751,-38.977,179.851,5.381,148.983
C05048=1219.592,-58.001,-38.965,179.849,5.381,148.983
C05049=1219.597,-58.250,-38.953,179.846,5.380,148.984
C05050=1219.602,-58.500,-38.940,179.844,5.380,148.985
C05051=1219.607,-58.749,-38.929,179.841,5.380,148.986
C05052=1219.613,-58.999,-38.917,179.839,5.380,148.986
C05053=1219.618,-59.249,-38.905,179.837,5.380,148.987
C05054=1219.623,-59.499,-38.893,179.834,5.380,148.988
C05055=1219.628,-59.748,-38.881,179.831,5.379,148.988
C05056=1219.633,-59.998,-38.869,179.829,5.380,148.989
C05057=1219.639,-60.248,-38.858,179.827,5.379,148.990
C05058=1219.643,-60.497,-38.846,179.825,5.380,148.991
C05059=1219.648,-60.747,-38.834,179.822,5.379,148.991
C05060=1219.654,-60.997,-38.822,179.820,5.379,148.992
C05061=1219.659,-61.247,-38.810,179.818,5.379,148.992
C05062=1219.664,-61.496,-38.798,179.815,5.378,148.993
C05063=1219.669,-61.746,-38.786,179.813,5.378,148.994
C05064=1219.675,-61.996,-38.774,179.810,5.378,148.995
C05065=1219.679,-62.245,-38.763,179.808,5.378,148.995
C05066=1219.684,-62.495,-38.750,179.805,5.378,148.996
C05067=1219.690,-62.745,-38.738,179.803,5.378,148.997
C05068=1219.694,-62.994,-38.727,179.801,5.378,148.997
C05069=1219.700,-63.244,-38.716,179.798,5.377,148.998
C05070=1219.706,-63.494,-38.704,179.796,5.378,148.999
C05071=1219.711,-63.743,-38.692,179.793,5.377,148.999
C05072=1219.716,-63.992,-38.680,179.791,5.378,149.000
C05073=1219.720,-64.242,-38.668,179.788,5.377,149.001
C05074=1219.726,-64.492,-38.657,179.786,5.377,149.002
C05075=1219.731,-64.742,-38.645,179.784,5.377,149.002
C05076=1219.736,-64.992,-38.633,179.781,5.376,149.003
C05077=1219.741,-65.242,-38.621,179.779,5.377,149.004
C05078=1219.747,-65.491,-38.610,179.776,5.376,149.004
C05079=1219.752,-65.741,-38.598,179.775,5.376,149.005
C05080=1219.757,-65.990,-38.586,179.772,5.376,149.006
C05081=1219.762,-66.239,-38.575,179.770,5.376,149.006
C05082=1219.767,-66.489,-38.563,179.767,5.376,149.007
C05083=1219.772,-66.739,-38.552,179.765,5.375,149.008
C05084=1219.778,-66.989,-38.540,179.763,5.376,149.008
C05085=1219.783,-67.239,-38.528,179.760,5.375,149.009
C05086=1219.788,-67.488,-38.517,179.758,5.376,149.010
C05087=1219.793,-67.738,-38.505,179.755,5.375,149.011
C05088=1219.798,-67.987,-38.494,179.753,5.375,149.011
C05089=1219.804,-68.237,-38.482,179.750,5.375,149.012
C05090=1219.808,-68.487,-38.471,179.748,5.375,149.013
C05091=1219.814,-68.737,-38.459,179.746,5.375,149.013
C05092=1219.819,-68.987,-38.447,179.743,5.374,149.014
C05093=1219.824,-69.236,-38.436,179.741,5.375,149.015
C05094=1219.829,-69.486,-38.424,179.738,5.374,149.015
C05095=1219.835,-69.735,-38.413,179.736,5.375,149.016
C05096=1219.840,-69.985,-38.401,179.734,5.374,149.017
C05097=1219.845,-70.235,-38.390,179.732,5.374,149.017
C05098=1219.850,-70.485,-38.378,179.729,5.374,149.018
C05099=1219.855,-70.734,-38.366,179.727,5.374,149.019
C05100=1219.861,-70.984,-38.355,179.724,5.374,149.020
C05101=1219.866,-71.233,-38.344,179.722,5.373,149.020
C05102=1219.871,-71.483,-38.332,179.720,5.374,149.021
C05103=1219.876,-71.733,-38.320,179.717,5.373,149.022
C05104=1219.881,-71.983,-38.308,179.715,5.373,149.022
C05105=1219.886,-72.232,-38.297,179.712,5.373,149.023
C05106=1219.892,-72.481,-38.286,179.710,5.373,149.024
C05107=1219.897,-72.731,-38.274,179.707,5.373,149.024
C05108=1219.902,-72.982,-38.263,179.705,5.373,149.025
C05109=1219.907,-73.231,-38.252,179.703,5.373,149.026
C05110=1219.912,-73.480,-38.241,179.700,5.372,149.027
C05111=1219.918,-73.730,-38.229,179.698,5.372,149.027
C05112=1219.923,-73.980,-38.218,179.696,5.372,149.028
C05113=1219.928,-74.230,-38.206,179.694,5.372,149.028
C05114=1219.934,-74.500,-38.194,179.691,5.372,149.029
C05115=1219.939,-74.770,-38.181,179.688,5.372,149.030
C05116=1219.944,-75.041,-38.169,179.686,5.372,149.031
C05117=1219.951,-75.311,-38.158,179.683,5.372,149.032
C05118=1219.956,-75.561,-38.146,179.681,5.372,149.032
C05119=1219.961,-75.811,-38.134,179.678,5.371,149.033
C05120=1219.965,-76.060,-38.123,179.676,5.372,149.034
C05121=1219.972,-76.310,-38.112,179.674,5.371,149.034
C05122=1219.976,-76.560,-38.101,179.671,5.371,149.035
C05123=1219.982,-76.810,-38.089,179.669,5.371,149.036
C05124=1219.987,-77.060,-38.078,179.667,5.370,149.036
C05125=1219.992,-77.308,-38.067,179.665,5.371,149.037
C05126=1219.998,-77.559,-38.056,179.662,5.370,149.038
C05127=1220.002,-77.809,-38.044,179.660,5.371,149.038
C05128=1220.008,-78.058,-38.034,179.657,5.370,149.039
C05129=1220.013,-78.308,-38.022,179.655,5.371,149.040
C05130=1220.018,-78.558,-38.011,179.652,5.370,149.041
C05131=1220.023,-78.808,-37.999,179.650,5.371,149.041
C05132=1220.029,-79.057,-37.988,179.648,5.370,149.042
C05133=1220.033,-79.306,-37.977,179.645,5.370,149.043
C05134=1220.038,-79.556,-37.966,179.643,5.370,149.043
C05135=1220.044,-79.806,-37.955,179.640,5.370,149.044
C05136=1220.049,-80.055,-37.944,179.638,5.370,149.045
C05137=1220.054,-80.306,-37.933,179.636,5.369,149.045
C05138=1220.060,-80.556,-37.921,179.634,5.369,149.046
C05139=1220.065,-80.804,-37.910,179.631,5.369,149.047
C05140=1220.070,-81.054,-37.899,179.629,5.369,149.047
C05141=1220.075,-81.305,-37.888,179.626,5.369,149.048
C05142=1220.081,-81.554,-37.877,179.624,5.369,149.049
C05143=1220.086,-81.804,-37.866,179.622,5.369,149.050
C05144=1220.090,-82.053,-37.855,179.619,5.369,149.050
C05145=1220.096,-82.303,-37.843,179.617,5.369,149.051
C05146=1220.101,-82.553,-37.833,179.615,5.369,149.052
C05147=1220.106,-82.803,-37.822,179.612,5.369,149.052
C05148=1220.111,-83.051,-37.811,179.610,5.369,149.053
C05149=1220.117,-83.302,-37.799,179.608,5.368,149.054
C05150=1220.122,-83.552,-37.788,179.606,5.369,149.054
C05151=1220.127,-83.801,-37.778,179.603,5.368,149.055
C05152=1220.132,-84.051,-37.767,179.601,5.368,149.056
C05153=1220.137,-84.301,-37.755,179.598,5.368,149.056
C05154=1220.143,-84.550,-37.745,179.596,5.368,149.057
C05155=1220.148,-84.800,-37.733,179.594,5.368,149.058
C05156=1220.153,-85.049,-37.723,179.591,5.367,149.059
C05157=1220.158,-85.299,-37.712,179.589,5.368,149.059
C05158=1220.164,-85.550,-37.701,179.586,5.367,149.060
C05159=1220.169,-85.799,-37.690,179.584,5.368,149.061
C05160=1220.174,-86.048,-37.678,179.582,5.367,149.061
C05161=1220.179,-86.298,-37.668,179.580,5.367,149.062
C05162=1220.184,-86.547,-37.657,179.577,5.367,149.063
C05163=1220.190,-86.798,-37.646,179.575,5.367,149.063
C05164=1220.195,-87.047,-37.635,179.572,5.367,149.064
C05165=1220.200,-87.297,-37.624,179.570,5.367,149.065
C05166=1220.205,-87.547,-37.613,179.568,5.367,149.065
C05167=1220.210,-87.796,-37.603,179.565,5.367,149.066
C05168=1220.215,-88.046,-37.591,179.563,5.367,149.067
C05169=1220.221,-88.296,-37.581,179.561,5.367,149.068
C05170=1220.226,-88.545,-37.569,179.558,5.366,149.068
C05171=1220.231,-88.796,-37.559,179.556,5.366,149.069
C05172=1220.236,-89.045,-37.548,179.554,5.366,149.069
C05173=1220.241,-89.295,-37.537,179.552,5.366,149.070
C05174=1220.247,-89.544,-37.527,179.549,5.366,149.071
C05175=1220.252,-89.794,-37.516,179.547,5.366,149.072
C05176=1220.257,-90.044,-37.505,179.544,5.366,149.072
C05177=1220.263,-90.293,-37.494,179.542,5.366,149.073
C05178=1220.268,-90.544,-37.483,179.539,5.366,149.074
C05179=1220.273,-90.793,-37.473,179.537,5.366,149.074
C05180=1220.278,-91.043,-37.462,179.535,5.365,149.075
C05181=1220.284,-91.292,-37.451,179.533,5.366,149.076
C05182=1220.288,-91.542,-37.440,179.530,5.365,149.076
C05183=1220.294,-91.792,-37.430,179.528,5.366,149.077
C05184=1220.299,-92.042,-37.419,179.526,5.365,149.078
C05185=1220.304,-92.291,-37.408,179.524,5.366,149.078
C05186=1220.309,-92.541,-37.398,179.521,5.365,149.079
C05187=1220.314,-92.791,-37.387,179.519,5.366,149.080
C05188=1220.319,-93.040,-37.376,179.516,5.365,149.081
C05189=1220.324,-93.290,-37.366,179.515,5.365,149.081
C05190=1220.330,-93.540,-37.354,179.512,5.365,149.082
C05191=1220.335,-93.790,-37.344,179.510,5.365,149.082
C05192=1220.341,-94.039,-37.333,179.507,5.365,149.083
C05193=1220.346,-94.290,-37.323,179.505,5.365,149.084
C05194=1220.351,-94.539,-37.312,179.502,5.364,149.085
C05195=1220.356,-94.789,-37.301,179.500,5.365,149.085
C05196=1220.362,-95.038,-37.291,179.498,5.364,149.086
C05197=1220.367,-95.288,-37.280,179.495,5.365,149.087
C05198=1220.372,-95.538,-37.270,179.493,5.364,149.087
C05199=1220.377,-95.788,-37.259,179.491,5.364,149.088
C05200=1220.383,-96.037,-37.249,179.488,5.364,149.089
C05201=1220.387,-96.287,-37.238,179.486,5.364,149.089
C05202=1220.393,-96.536,-37.227,179.484,5.364,149.090
C05203=1220.398,-96.787,-37.217,179.482,5.364,149.091
C05204=1220.404,-97.036,-37.207,179.479,5.364,149.092
C05205=1220.409,-97.285,-37.196,179.477,5.364,149.092
C05206=1220.414,-97.535,-37.185,179.475,5.363,149.093
C05207=1220.420,-97.785,-37.175,179.473,5.364,149.093
C05208=1220.425,-98.035,-37.164,179.470,5.363,149.094
C05209=1220.430,-98.285,-37.154,179.468,5.364,149.095
C05210=1220.435,-98.534,-37.143,179.465,5.363,149.096
C05211=1220.440,-98.784,-37.133,179.463,5.364,149.096
C05212=1220.445,-99.034,-37.123,179.460,5.363,149.097
C05213=1220.450,-99.283,-37.112,179.458,5.363,149.098
C05214=1220.455,-99.534,-37.102,179.456,5.363,149.098
C05215=1220.461,-99.783,-37.091,179.454,5.363,149.099
C05216=1220.466,-100.032,-37.081,179.451,5.363,149.100
C05217=1220.471,-100.282,-37.070,179.449,5.363,149.100
C05218=1220.476,-100.554,-37.059,179.447,5.363,149.101
C05219=1220.483,-100.825,-37.048,179.444,5.362,149.102
C05220=1220.488,-101.095,-37.036,179.442,5.362,149.102
C05221=1220.494,-101.367,-37.025,179.439,5.362,149.103
C05222=1220.499,-101.616,-37.015,179.437,5.362,149.104
C05223=1220.504,-101.867,-37.004,179.434,5.362,149.105
C05224=1220.510,-102.116,-36.994,179.432,5.362,149.105
C05225=1220.515,-102.365,-36.984,179.430,5.362,149.106
C05226=1220.520,-102.616,-36.974,179.427,5.362,149.107
C05227=1220.525,-102.865,-36.963,179.425,5.362,149.107
C05228=1220.530,-103.115,-36.953,179.423,5.362,149.108
C05229=1220.536,-103.365,-36.943,179.421,5.361,149.109
C05230=1220.541,-103.614,-36.932,179.418,5.362,149.109
C05231=1220.546,-103.864,-36.921,179.416,5.361,149.110
C05232=1220.551,-104.113,-36.912,179.414,5.362,149.111
C05233=1220.557,-104.363,-36.901,179.411,5.361,149.112
C05234=1220.562,-104.613,-36.891,179.409,5.362,149.112
C05235=1220.567,-104.863,-36.881,179.406,5.361,149.113
C05236=1220.572,-105.113,-36.870,179.405,5.361,149.113
C05237=1220.577,-105.362,-36.860,179.402,5.361,149.114
C05238=1220.583,-105.612,-36.850,179.400,5.361,149.115
C05239=1220.588,-105.862,-36.840,179.398,5.362,149.116
C05240=1220.593,-106.112,-36.829,179.395,5.361,149.116
C05241=1220.599,-106.361,-36.819,179.393,5.362,149.117
C05242=1220.603,-106.611,-36.809,179.391,5.361,149.117
C05243=1220.609,-106.861,-36.799,179.389,5.361,149.118
C05244=1220.614,-107.110,-36.789,179.386,5.361,149.119
C05245=1220.619,-107.360,-36.778,179.384,5.361,149.120
C05246=1220.625,-107.610,-36.768,179.381,5.361,149.120
C05247=1220.630,-107.860,-36.759,179.379,5.361,149.121
C05248=1220.635,-108.110,-36.749,179.377,5.361,149.122
C05249=1220.641,-108.360,-36.738,179.375,5.361,149.122
C05250=1220.646,-108.609,-36.728,179.372,5.360,149.123
C05251=1220.651,-108.859,-36.718,179.370,5.361,149.124
C05252=1220.656,-109.109,-36.708,179.367,5.360,149.124
C05253=1220.662,-109.358,-36.698,179.365,5.360,149.125
C05254=1220.667,-109.608,-36.687,179.363,5.360,149.126
C05255=1220.672,-109.858,-36.678,179.361,5.360,149.126
C05256=1220.677,-110.107,-36.667,179.358,5.360,149.127
C05257=1220.682,-110.357,-36.657,179.356,5.360,149.128
C05258=1220.687,-110.607,-36.648,179.354,5.360,149.128
C05259=1220.693,-110.857,-36.638,179.352,5.360,149.129
C05260=1220.699,-111.106,-36.627,179.349,5.360,149.130
C05261=1220.704,-111.357,-36.617,179.347,5.360,149.130
C05262=1220.708,-111.606,-36.607,179.345,5.360,149.131
C05263=1220.714,-111.855,-36.597,179.343,5.359,149.132
C05264=1220.719,-112.106,-36.587,179.340,5.360,149.133
C05265=1220.724,-112.355,-36.578,179.338,5.359,149.133
C05266=1220.730,-112.605,-36.567,179.336,5.360,149.134
C05267=1220.735,-112.854,-36.557,179.333,5.359,149.134
C05268=1220.740,-113.104,-36.547,179.331,5.359,149.135
C05269=1220.745,-113.354,-36.537,179.329,5.359,149.136
C05270=1220.751,-113.604,-36.527,179.327,5.359,149.137
C05271=1220.756,-113.853,-36.518,179.324,5.359,149.137
C05272=1220.761,-114.104,-36.507,179.322,5.359,149.138
C05273=1220.767,-114.353,-36.497,179.320,5.358,149.138
C05274=1220.772,-114.603,-36.488,179.318,5.359,149.139
C05275=1220.777,-114.853,-36.478,179.315,5.359,149.140
C05276=1220.782,-115.103,-36.467,179.313,5.359,149.141
C05277=1220.787,-115.352,-36.458,179.311,5.359,149.141
C05278=1220.793,-115.602,-36.448,179.309,5.358,149.142
C05279=1220.798,-115.851,-36.439,179.306,5.359,149.143
C05280=1220.803,-116.102,-36.428,179.304,5.358,149.143
C05281=1220.809,-116.351,-36.418,179.302,5.359,149.144
C05282=1220.814,-116.601,-36.409,179.299,5.358,149.145
C05283=1220.819,-116.851,-36.399,179.297,5.358,149.145
C05284=1220.824,-117.100,-36.389,179.295,5.358,149.146
C05285=1220.830,-117.351,-36.379,179.293,5.358,149.147
C05286=1220.835,-117.600,-36.369,179.290,5.358,149.147
C05287=1220.840,-117.849,-36.359,179.288,5.358,149.148
C05288=1220.846,-118.100,-36.350,179.286,5.358,149.149
C05289=1220.851,-118.349,-36.340,179.284,5.358,149.149
C05290=1220.856,-118.599,-36.330,179.281,5.358,149.150
C05291=1220.861,-118.849,-36.321,179.279,5.358,149.151
C05292=1220.867,-119.098,-36.311,179.277,5.358,149.151
C05293=1220.871,-119.348,-36.301,179.274,5.358,149.152
C05294=1220.877,-119.598,-36.292,179.272,5.358,149.153
C05295=1220.882,-119.848,-36.282,179.270,5.357,149.153
C05296=1220.887,-120.097,-36.271,179.268,5.358,149.154
C05297=1220.893,-120.348,-36.262,179.265,5.357,149.155
C05298=1220.898,-120.597,-36.252,179.263,5.357,149.155
C05299=1220.904,-120.847,-36.243,179.261,5.357,149.156
C05300=1220.909,-121.096,-36.233,179.259,5.357,149.157
C05301=1220.914,-121.346,-36.223,179.256,5.358,149.157
C05302=1220.919,-121.596,-36.214,179.254,5.357,149.158
C05303=1220.924,-121.846,-36.203,179.252,5.357,149.159
C05304=1220.930,-122.096,-36.195,179.250,5.357,149.159
C05305=1220.935,-122.345,-36.184,179.247,5.357,149.160
C05306=1220.940,-122.595,-36.175,179.245,5.357,149.161
C05307=1220.945,-122.844,-36.166,179.243,5.357,149.161
C05308=1220.951,-123.095,-36.156,179.240,5.356,149.162
C05309=1220.955,-123.344,-36.146,179.238,5.357,149.163
C05310=1220.961,-123.594,-36.136,179.236,5.356,149.163
C05311=1220.966,-123.844,-36.127,179.234,5.357,149.164
C05312=1220.972,-124.093,-36.117,179.232,5.357,149.165
C05313=1220.977,-124.343,-36.108,179.229,5.356,149.165
C05314=1220.983,-124.593,-36.098,179.227,5.357,149.166
C05315=1220.988,-124.843,-36.089,179.225,5.356,149.167
C05316=1220.993,-125.093,-36.079,179.222,5.357,149.167
C05317=1220.998,-125.343,-36.070,179.220,5.356,149.168
C05318=1221.003,-125.593,-36.061,179.218,5.356,149.169
C05319=1221.009,-125.842,-36.051,179.215,5.356,149.169
C05320=1221.014,-126.092,-36.042,179.213,5.356,149.170
C05321=1221.019,-126.341,-36.031,179.211,5.357,149.171
C05322=1220.598,-126.352,-36.068,179.207,5.360,149.173
C05323=1220.592,-126.103,-36.078,179.209,5.359,149.172
C05324=1220.587,-125.853,-36.087,179.212,5.359,149.171
C05325=1220.581,-125.603,-36.097,179.214,5.360,149.171
C05326=1220.577,-125.353,-36.106,179.216,5.359,149.170
C05327=1220.572,-125.103,-36.116,179.218,5.360,149.169
C05328=1220.566,-124.853,-36.125,179.221,5.359,149.169
C05329=1220.561,-124.604,-36.135,179.223,5.360,149.168
C05330=1220.555,-124.354,-36.145,179.225,5.360,149.167
C05331=1220.550,-124.105,-36.154,179.228,5.360,149.167
C05332=1220.544,-123.855,-36.164,179.230,5.360,149.166
C05333=1220.540,-123.605,-36.173,179.231,5.360,149.165
C05334=1220.534,-123.355,-36.183,179.234,5.360,149.165
C05335=1220.529,-123.105,-36.193,179.236,5.360,149.164
C05336=1220.524,-122.855,-36.202,179.239,5.360,149.163
C05337=1220.519,-122.606,-36.212,179.241,5.360,149.163
C05338=1220.513,-122.356,-36.221,179.243,5.361,149.162
C05339=1220.508,-122.106,-36.231,179.245,5.360,149.161
C05340=1220.503,-121.857,-36.240,179.248,5.361,149.161
C05341=1220.497,-121.607,-36.250,179.250,5.360,149.160
C05342=1220.493,-121.357,-36.260,179.253,5.361,149.159
C05343=1220.487,-121.107,-36.270,179.254,5.361,149.159
C05344=1220.482,-120.858,-36.279,179.256,5.360,149.158
C05345=1220.476,-120.607,-36.289,179.259,5.361,149.157
C05346=1220.471,-120.358,-36.298,179.261,5.360,149.157
C05347=1220.466,-120.109,-36.308,179.264,5.361,149.156
C05348=1220.461,-119.858,-36.318,179.265,5.361,149.155
C05349=1220.456,-119.609,-36.328,179.268,5.361,149.155
C05350=1220.450,-119.359,-36.337,179.270,5.361,149.154
C05351=1220.445,-119.109,-36.347,179.273,5.361,149.153
C05352=1220.439,-118.860,-36.357,179.274,5.361,149.153
C05353=1220.434,-118.610,-36.366,179.277,5.362,149.152
C05354=1220.429,-118.360,-36.377,179.279,5.361,149.151
C05355=1220.424,-118.110,-36.386,179.282,5.362,149.151
C05356=1220.418,-117.860,-36.396,179.284,5.361,149.150
C05357=1220.413,-117.611,-36.405,179.286,5.361,149.149
C05358=1220.408,-117.361,-36.416,179.288,5.362,149.149
C05359=1220.403,-117.111,-36.425,179.290,5.361,149.148
C05360=1220.398,-116.861,-36.435,179.293,5.362,149.147
C05361=1220.392,-116.612,-36.445,179.295,5.361,149.147
C05362=1220.387,-116.362,-36.454,179.298,5.362,149.146
C05363=1220.382,-116.112,-36.465,179.299,5.362,149.145
C05364=1220.377,-115.862,-36.474,179.302,5.362,149.145
C05365=1220.371,-115.613,-36.485,179.304,5.362,149.144
C05366=1220.366,-115.363,-36.494,179.307,5.362,149.143
C05367=1220.361,-115.114,-36.504,179.309,5.362,149.143
C05368=1220.356,-114.863,-36.514,179.311,5.363,149.142
C05369=1220.350,-114.613,-36.524,179.313,5.362,149.141
C05370=1220.345,-114.364,-36.533,179.315,5.362,149.141
C05371=1220.339,-114.114,-36.544,179.318,5.362,149.140
C05372=1220.335,-113.864,-36.554,179.320,5.362,149.139
C05373=1220.329,-113.615,-36.564,179.322,5.363,149.139
C05374=1220.324,-113.365,-36.573,179.324,5.362,149.138
C05375=1220.319,-113.115,-36.583,179.327,5.363,149.137
C05376=1220.314,-112.865,-36.593,179.329,5.363,149.137
C05377=1220.308,-112.616,-36.604,179.332,5.363,149.136
C05378=1220.303,-112.366,-36.613,179.334,5.363,149.135
C05379=1220.297,-112.116,-36.623,179.336,5.363,149.135
C05380=1220.292,-111.866,-36.633,179.338,5.363,149.134
C05381=1220.287,-111.617,-36.643,179.341,5.363,149.133
C05382=1220.282,-111.367,-36.653,179.343,5.363,149.132
C05383=1220.277,-111.117,-36.664,179.346,5.363,149.132
C05384=1220.271,-110.867,-36.674,179.348,5.363,149.131
C05385=1220.266,-110.618,-36.683,179.349,5.363,149.131
C05386=1220.260,-110.368,-36.693,179.352,5.364,149.130
C05387=1220.255,-110.118,-36.704,179.354,5.363,149.129
C05388=1220.251,-109.869,-36.713,179.357,5.364,149.128
C05389=1220.245,-109.619,-36.723,179.359,5.363,149.128
C05390=1220.240,-109.369,-36.734,179.361,5.364,149.127
C05391=1220.234,-109.119,-36.744,179.363,5.364,149.127
C05392=1220.230,-108.870,-36.754,179.366,5.364,149.126
C05393=1220.224,-108.619,-36.764,179.368,5.364,149.125
C05394=1220.219,-108.370,-36.774,179.370,5.364,149.124
C05395=1220.213,-108.120,-36.784,179.373,5.364,149.124
C05396=1220.208,-107.871,-36.794,179.375,5.364,149.123
C05397=1220.203,-107.621,-36.804,179.377,5.364,149.122
C05398=1220.198,-107.371,-36.815,179.380,5.365,149.122
C05399=1220.192,-107.122,-36.825,179.382,5.364,149.121
C05400=1220.188,-106.872,-36.835,179.384,5.365,149.120
C05401=1220.182,-106.622,-36.845,179.386,5.364,149.120
C05402=1220.177,-106.372,-36.856,179.389,5.365,149.119
C05403=1220.172,-106.122,-36.866,179.391,5.365,149.118
C05404=1220.166,-105.873,-36.876,179.393,5.365,149.118
C05405=1220.162,-105.623,-36.886,179.395,5.365,149.117
C05406=1220.156,-105.373,-36.896,179.398,5.364,149.116
C05407=1220.151,-105.124,-36.906,179.400,5.365,149.116
C05408=1220.146,-104.873,-36.917,179.402,5.364,149.115
C05409=1220.140,-104.624,-36.927,179.405,5.365,149.114
C05410=1220.135,-104.375,-36.937,179.407,5.365,149.114
C05411=1220.130,-104.124,-36.947,179.409,5.365,149.113
C05412=1220.124,-103.875,-36.958,179.411,5.365,149.112
C05413=1220.119,-103.625,-36.968,179.414,5.365,149.111
C05414=1220.114,-103.375,-36.978,179.416,5.365,149.111
C05415=1220.108,-103.126,-36.989,179.419,5.365,149.110
C05416=1220.104,-102.876,-36.998,179.421,5.365,149.109
C05417=1220.098,-102.626,-37.009,179.423,5.366,149.109
C05418=1220.093,-102.376,-37.019,179.425,5.365,149.108
C05419=1220.088,-102.126,-37.029,179.428,5.366,149.107
C05420=1220.083,-101.877,-37.040,179.430,5.366,149.107
C05421=1220.078,-101.627,-37.051,179.433,5.366,149.106
C05422=1220.072,-101.378,-37.061,179.435,5.366,149.105
C05423=1220.067,-101.106,-37.072,179.437,5.366,149.105
C05424=1220.061,-100.835,-37.084,179.439,5.366,149.104
C05425=1220.055,-100.564,-37.094,179.442,5.366,149.103
C05426=1220.049,-100.293,-37.106,179.445,5.366,149.102
C05427=1220.045,-100.044,-37.116,179.447,5.366,149.102
C05428=1220.040,-99.794,-37.127,179.450,5.367,149.101
C05429=1220.034,-99.544,-37.137,179.452,5.366,149.100
C05430=1220.029,-99.294,-37.147,179.454,5.367,149.100
C05431=1220.023,-99.044,-37.158,179.456,5.367,149.099
C05432=1220.019,-98.795,-37.169,179.459,5.367,149.098
C05433=1220.013,-98.545,-37.179,179.461,5.367,149.098
C05434=1220.008,-98.295,-37.190,179.463,5.367,149.097
C05435=1220.002,-98.045,-37.200,179.465,5.367,149.096
C05436=1219.997,-97.796,-37.210,179.468,5.367,149.096
C05437=1219.992,-97.546,-37.221,179.470,5.367,149.095
C05438=1219.987,-97.297,-37.232,179.473,5.367,149.094
C05439=1219.982,-97.046,-37.242,179.474,5.367,149.094
C05440=1219.976,-96.797,-37.252,179.477,5.368,149.093
C05441=1219.971,-96.547,-37.263,179.479,5.367,149.092
C05442=1219.966,-96.298,-37.274,179.482,5.368,149.091
C05443=1219.961,-96.047,-37.285,179.484,5.367,149.091
C05444=1219.955,-95.798,-37.295,179.487,5.368,149.090
C05445=1219.950,-95.548,-37.305,179.489,5.367,149.089
C05446=1219.945,-95.299,-37.316,179.491,5.368,149.089
C05447=1219.940,-95.048,-37.327,179.493,5.368,149.088
C05448=1219.934,-94.799,-37.337,179.496,5.368,149.087
C05449=1219.930,-94.549,-37.348,179.498,5.368,149.087
C05450=1219.924,-94.300,-37.359,179.501,5.368,149.086
C05451=1219.919,-94.050,-37.369,179.503,5.368,149.085
C05452=1219.913,-93.800,-37.379,179.505,5.368,149.085
C05453=1219.909,-93.550,-37.391,179.507,5.368,149.084
C05454=1219.903,-93.301,-37.401,179.510,5.369,149.083
C05455=1219.898,-93.051,-37.411,179.512,5.369,149.083
C05456=1219.893,-92.802,-37.422,179.514,5.369,149.082
C05457=1219.888,-92.551,-37.433,179.516,5.369,149.081
C05458=1219.882,-92.302,-37.443,179.519,5.369,149.081
C05459=1219.877,-92.052,-37.454,179.521,5.369,149.080
C05460=1219.872,-91.803,-37.465,179.524,5.369,149.079
C05461=1219.867,-91.553,-37.476,179.526,5.369,149.078
C05462=1219.862,-91.304,-37.486,179.529,5.369,149.078
C05463=1219.856,-91.053,-37.497,179.531,5.369,149.077
C05464=1219.851,-90.803,-37.509,179.533,5.370,149.077
C05465=1219.846,-90.554,-37.519,179.535,5.369,149.076
C05466=1219.841,-90.304,-37.530,179.538,5.370,149.075
C05467=1219.835,-90.055,-37.540,179.540,5.369,149.074
C05468=1219.830,-89.804,-37.551,179.542,5.370,149.074
C05469=1219.825,-89.555,-37.562,179.544,5.369,149.073
C05470=1219.820,-89.305,-37.572,179.547,5.370,149.072
C05471=1219.815,-89.056,-37.583,179.549,5.370,149.072
C05472=1219.810,-88.806,-37.594,179.552,5.370,149.071
C05473=1219.804,-88.556,-37.606,179.554,5.370,149.070
C05474=1219.799,-88.307,-37.616,179.556,5.370,149.070
C05475=1219.794,-88.057,-37.627,179.558,5.370,149.069
C05476=1219.788,-87.807,-37.637,179.561,5.371,149.068
C05477=1219.783,-87.557,-37.648,179.563,5.370,149.068
C05478=1219.779,-87.308,-37.659,179.566,5.371,149.067
C05479=1219.772,-87.058,-37.670,179.568,5.370,149.066
C05480=1219.768,-86.808,-37.681,179.570,5.371,149.065
C05481=1219.762,-86.558,-37.692,179.573,5.370,149.065
C05482=1219.757,-86.309,-37.703,179.575,5.371,149.064
C05483=1219.753,-86.059,-37.714,179.577,5.371,149.063
C05484=1219.747,-85.810,-37.724,179.580,5.371,149.063
